LIN {X 0,Y 417.78,Z 272.398,A -85,B 0,C 180,E1 -10353.858,E2 -10353.858} C_VEL
LIN {X 0,Y 417.736,Z 275.155,A -85,B 0,C 180,E1 -10356.981,E2 -10356.981} C_VEL
LIN {X 0,Y 417.624,Z 276.659,A -85,B 0,C 180,E1 -10358.65,E2 -10358.65} C_VEL
LIN {X 0,Y 420.264,Z 284.393,A -85,B 0,C 180,E1 -10359.007,E2 -10359.007} C_VEL
LIN {X 0,Y 425.304,Z 299.305,A -85,B 0,C 180,E1 -10359.798,E2 -10359.798} C_VEL
LIN {X 0,Y 427.282,Z 306.519,A -85,B 0,C 180,E1 -10360.222,E2 -10360.222} C_VEL
LIN {X 0,Y 427.662,Z 310.082,A -85,B 0,C 180,E1 -10360.409,E2 -10360.409} C_VEL
LIN {X 0,Y 426.563,Z 315.588,A -85,B 0,C 180,E1 -10360.631,E2 -10360.631} C_VEL
LIN {X 0,Y 420.151,Z 329.943,A -85,B 0,C 180,E1 -10361.176,E2 -10361.176} C_VEL
LIN {X 0,Y 419.11,Z 333.547,A -85,B 0,C 180,E1 -10361.385,E2 -10361.385} C_VEL
LIN {X 0,Y 418.867,Z 335.334,A -85,B 0,C 180,E1 -10361.51,E2 -10361.51} C_VEL
LIN {X 0,Y 417.7,Z 349.15,A -85,B 0,C 180,E1 -10362.634,E2 -10362.634} C_VEL
LIN {X 0,Y 416.435,Z 362.009,A -85,B 0,C 180,E1 -10363.915,E2 -10363.915} C_VEL
LIN {X 0,Y 415.171,Z 374.509,A -85,B 0,C 180,E1 -10365.434,E2 -10365.434} C_VEL
LIN {X 0,Y 413.977,Z 385.392,A -85,B 0,C 180,E1 -10367.028,E2 -10367.028} C_VEL
LIN {X 0,Y 412.925,Z 394.448,A -85,B 0,C 180,E1 -10368.609,E2 -10368.609} C_VEL
LIN {X 0,Y 412.129,Z 402.506,A -85,B 0,C 180,E1 -10370.301,E2 -10370.301} C_VEL
LIN {X 0,Y 411.345,Z 410.582,A -85,B 0,C 180,E1 -10372.365,E2 -10372.365} C_VEL
LIN {X 0,Y 410.794,Z 416.403,A -85,B 0,C 180,E1 -10374.242,E2 -10374.242} C_VEL
LIN {X 0,Y 410.419,Z 421.643,A -85,B 0,C 180,E1 -10376.437,E2 -10376.437} C_VEL
LIN {X 0,Y 410.248,Z 423.698,A -85,B 0,C 180,E1 -10377.55,E2 -10377.55} C_VEL
LIN {X 0,Y 410.052,Z 425.834,A -85,B 0,C 180,E1 -10379.065,E2 -10379.065} C_VEL
LIN {X 0,Y 409.943,Z 427.623,A -85,B 0,C 180,E1 -10381.001,E2 -10381.001} C_VEL
LIN {X 0,Y 409.913,Z 428.276,A -85,B 0,C 180,E1 -10382.851,E2 -10382.851} C_VEL
LIN {X 0,Y 409.904,Z 427.963,A -85,B 0,C 180,E1 -10384.618,E2 -10384.618} C_VEL
LIN {X 0,Y 410.045,Z 426.269,A -85,B 0,C 180,E1 -10386.861,E2 -10386.861} C_VEL
LIN {X 0,Y 410.294,Z 423.778,A -85,B 0,C 180,E1 -10388.697,E2 -10388.697} C_VEL
LIN {X 0,Y 410.587,Z 420.138,A -85,B 0,C 180,E1 -10390.574,E2 -10390.574} C_VEL
LIN {X 0,Y 411.1,Z 414.621,A -85,B 0,C 180,E1 -10392.686,E2 -10392.686} C_VEL
LIN {X 0,Y 411.744,Z 407.684,A -85,B 0,C 180,E1 -10394.737,E2 -10394.737} C_VEL
LIN {X 0,Y 412.525,Z 400.757,A -85,B 0,C 180,E1 -10396.389,E2 -10396.389} C_VEL
LIN {X 0,Y 413.456,Z 392.475,A -85,B 0,C 180,E1 -10398.043,E2 -10398.043} C_VEL
LIN {X 0,Y 414.566,Z 382.455,A -85,B 0,C 180,E1 -10399.717,E2 -10399.717} C_VEL
LIN {X 0,Y 415.656,Z 372.901,A -85,B 0,C 180,E1 -10401.056,E2 -10401.056} C_VEL
LIN {X 0,Y 416.904,Z 361.556,A -85,B 0,C 180,E1 -10402.4,E2 -10402.4} C_VEL
LIN {X 0,Y 418.204,Z 348.685,A -85,B 0,C 180,E1 -10403.665,E2 -10403.665} C_VEL
LIN {X 0,Y 419.338,Z 335.97,A -85,B 0,C 180,E1 -10404.694,E2 -10404.694} C_VEL
LIN {X 0,Y 420.418,Z 322.342,A -85,B 0,C 180,E1 -10405.583,E2 -10405.583} C_VEL
LIN {X 0,Y 421.137,Z 309.245,A -85,B 0,C 180,E1 -10406.263,E2 -10406.263} C_VEL
LIN {X 0,Y 417.181,Z 296.351,A -85,B 0,C 180,E1 -10407.067,E2 -10407.067} C_VEL
LIN {X 0,Y 411.697,Z 281.87,A -85,B 0,C 180,E1 -10407.87,E2 -10407.87} C_VEL
LIN {X 0,Y 410.707,Z 278.898,A -85,B 0,C 180,E1 -10408.024,E2 -10408.024} C_VEL
LIN {X 0,Y 410.788,Z 276.178,A -85,B 0,C 180,E1 -10411.379,E2 -10411.379} C_VEL
LIN {X 0,Y 410.912,Z 273.548,A -85,B 0,C 180,E1 -10414.687,E2 -10414.687} C_VEL
LIN {X 0,Y 411.031,Z 271.058,A -85,B 0,C 180,E1 -10417.905,E2 -10417.905} C_VEL
LIN {X 0,Y 411.105,Z 269.368,A -85,B 0,C 180,E1 -10420.09,E2 -10420.09} C_VEL
LIN {X 0,Y 411.104,Z 268.906,A -85,B 0,C 180,E1 -10421.047,E2 -10421.047} C_VEL
LIN {X 0,Y 411.247,Z 268.889,A -85,B 0,C 180,E1 -10424.133,E2 -10424.133} C_VEL
LIN {X 0,Y 411.296,Z 268.878,A -85,B 0,C 180,E1 -10427.167,E2 -10427.167} C_VEL
LIN {X 0,Y 411.287,Z 268.881,A -85,B 0,C 180,E1 -10430.162,E2 -10430.162} C_VEL
LIN {X 0,Y 411.455,Z 268.86,A -85,B 0,C 180,E1 -10433.134,E2 -10433.134} C_VEL
LIN {X 0,Y 411.308,Z 268.879,A -85,B 0,C 180,E1 -10435.1,E2 -10435.1} C_VEL
LIN {X 0,Y 411.509,Z 268.851,A -85,B 0,C 180,E1 -10438.044,E2 -10438.044} C_VEL
LIN {X 0,Y 411.637,Z 268.834,A -85,B 0,C 180,E1 -10440.001,E2 -10440.001} C_VEL
LIN {X 0,Y 411.462,Z 268.859,A -85,B 0,C 180,E1 -10442.938,E2 -10442.938} C_VEL
LIN {X 0,Y 411.457,Z 268.859,A -85,B 0,C 180,E1 -10446.868,E2 -10446.868} C_VEL
LIN {X 0,Y 411.29,Z 268.88,A -85,B 0,C 180,E1 -10449.84,E2 -10449.84} C_VEL
LIN {X 0,Y 411.302,Z 268.875,A -85,B 0,C 180,E1 -10453.105,E2 -10453.105} C_VEL
LIN {X 0,Y 411.254,Z 268.882,A -85,B 0,C 180,E1 -10456.89,E2 -10456.89} C_VEL
LIN {X 0,Y 411.228,Z 268.886,A -85,B 0,C 180,E1 -10459.988,E2 -10459.988} C_VEL
LIN {X 0,Y 411.201,Z 268.89,A -85,B 0,C 180,E1 -10463.148,E2 -10463.148} C_VEL
LIN {X 0,Y 411.236,Z 268.888,A -85,B 0,C 180,E1 -10466.382,E2 -10466.382} C_VEL
LIN {X 0,Y 411.198,Z 268.895,A -85,B 0,C 180,E1 -10469.714,E2 -10469.714} C_VEL
LIN {X 0,Y 411.204,Z 268.899,A -85,B 0,C 180,E1 -10473.157,E2 -10473.157} C_VEL
LIN {X 0,Y 411.191,Z 268.898,A -85,B 0,C 180,E1 -10476.553,E2 -10476.553} C_VEL
LIN {X 0,Y 411.228,Z 269.052,A -85,B 0,C 180,E1 -10478.174,E2 -10478.174} C_VEL
LIN {X 0,Y 411.775,Z 272.063,A -85,B 0,C 180,E1 -10480.434,E2 -10480.434} C_VEL
LIN {X 0,Y 412.581,Z 276.778,A -85,B 0,C 180,E1 -10483.622,E2 -10483.622} C_VEL
LIN {X 0,Y 413.264,Z 280.257,A -85,B 0,C 180,E1 -10485.794,E2 -10485.794} C_VEL
LIN {X 0,Y 413.665,Z 283.769,A -85,B 0,C 180,E1 -10487.835,E2 -10487.835} C_VEL
LIN {X 0,Y 413.41,Z 288.694,A -85,B 0,C 180,E1 -10490.455,E2 -10490.455} C_VEL
LIN {X 0,Y 412.873,Z 294.663,A -85,B 0,C 180,E1 -10493.433,E2 -10493.433} C_VEL
LIN {X 0,Y 412.345,Z 302.105,A -85,B 0,C 180,E1 -10496.948,E2 -10496.948} C_VEL
LIN {X 0,Y 411.837,Z 310.013,A -85,B 0,C 180,E1 -10500.496,E2 -10500.496} C_VEL
LIN {X 0,Y 411.424,Z 317.27,A -85,B 0,C 180,E1 -10503.633,E2 -10503.633} C_VEL
LIN {X 0,Y 411.288,Z 320.498,A -85,B 0,C 180,E1 -10505.002,E2 -10505.002} C_VEL
LIN {X 0,Y 415.679,Z 338.456,A -85,B 0,C 180,E1 -10505.742,E2 -10505.742} C_VEL
LIN {X 0,Y 418.813,Z 353.128,A -85,B 0,C 180,E1 -10506.502,E2 -10506.502} C_VEL
LIN {X 0,Y 420.119,Z 360.598,A -85,B 0,C 180,E1 -10506.938,E2 -10506.938} C_VEL
LIN {X 0,Y 419.113,Z 374.52,A -85,B 0,C 180,E1 -10507.705,E2 -10507.705} C_VEL
LIN {X 0,Y 417.815,Z 388.486,A -85,B 0,C 180,E1 -10508.67,E2 -10508.67} C_VEL
LIN {X 0,Y 416.538,Z 401.32,A -85,B 0,C 180,E1 -10509.765,E2 -10509.765} C_VEL
LIN {X 0,Y 415.192,Z 414.332,A -85,B 0,C 180,E1 -10511.112,E2 -10511.112} C_VEL
LIN {X 0,Y 414.139,Z 425.261,A -85,B 0,C 180,E1 -10512.47,E2 -10512.47} C_VEL
LIN {X 0,Y 412.996,Z 435.377,A -85,B 0,C 180,E1 -10513.948,E2 -10513.948} C_VEL
LIN {X 0,Y 411.994,Z 445.292,A -85,B 0,C 180,E1 -10515.68,E2 -10515.68} C_VEL
LIN {X 0,Y 411.241,Z 453.581,A -85,B 0,C 180,E1 -10517.415,E2 -10517.415} C_VEL
LIN {X 0,Y 410.766,Z 460.444,A -85,B 0,C 180,E1 -10519.153,E2 -10519.153} C_VEL
LIN {X 0,Y 410.323,Z 466.793,A -85,B 0,C 180,E1 -10521.133,E2 -10521.133} C_VEL
LIN {X 0,Y 410.163,Z 471.718,A -85,B 0,C 180,E1 -10523.112,E2 -10523.112} C_VEL
LIN {X 0,Y 410.032,Z 475.329,A -85,B 0,C 180,E1 -10525.084,E2 -10525.084} C_VEL
LIN {X 0,Y 410.002,Z 477.711,A -85,B 0,C 180,E1 -10527.053,E2 -10527.053} C_VEL
LIN {X 0,Y 409.917,Z 478.915,A -85,B 0,C 180,E1 -10529.018,E2 -10529.018} C_VEL
LIN {X 0,Y 409.917,Z 478.931,A -85,B 0,C 180,E1 -10530.983,E2 -10530.983} C_VEL
LIN {X 0,Y 409.987,Z 477.754,A -85,B 0,C 180,E1 -10532.948,E2 -10532.948} C_VEL
LIN {X 0,Y 410.027,Z 475.402,A -85,B 0,C 180,E1 -10534.917,E2 -10534.917} C_VEL
LIN {X 0,Y 410.159,Z 471.832,A -85,B 0,C 180,E1 -10536.89,E2 -10536.89} C_VEL
LIN {X 0,Y 410.324,Z 466.949,A -85,B 0,C 180,E1 -10538.868,E2 -10538.868} C_VEL
LIN {X 0,Y 410.763,Z 460.638,A -85,B 0,C 180,E1 -10540.849,E2 -10540.849} C_VEL
LIN {X 0,Y 411.293,Z 453.823,A -85,B 0,C 180,E1 -10542.584,E2 -10542.584} C_VEL
LIN {X 0,Y 412,Z 445.583,A -85,B 0,C 180,E1 -10544.321,E2 -10544.321} C_VEL
LIN {X 0,Y 413.025,Z 435.723,A -85,B 0,C 180,E1 -10546.053,E2 -10546.053} C_VEL
LIN {X 0,Y 414.16,Z 425.652,A -85,B 0,C 180,E1 -10547.531,E2 -10547.531} C_VEL
LIN {X 0,Y 415.348,Z 413.696,A -85,B 0,C 180,E1 -10549.01,E2 -10549.01} C_VEL
LIN {X 0,Y 416.611,Z 401.802,A -85,B 0,C 180,E1 -10550.233,E2 -10550.233} C_VEL
LIN {X 0,Y 417.807,Z 388.969,A -85,B 0,C 180,E1 -10551.332,E2 -10551.332} C_VEL
LIN {X 0,Y 419.125,Z 375.006,A -85,B 0,C 180,E1 -10552.296,E2 -10552.296} C_VEL
LIN {X 0,Y 420.22,Z 360.344,A -85,B 0,C 180,E1 -10553.095,E2 -10553.095} C_VEL
LIN {X 0,Y 416.994,Z 344.752,A -85,B 0,C 180,E1 -10553.963,E2 -10553.963} C_VEL
LIN {X 0,Y 413.283,Z 329.145,A -85,B 0,C 180,E1 -10554.659,E2 -10554.659} C_VEL
LIN {X 0,Y 411.317,Z 321.374,A -85,B 0,C 180,E1 -10554.967,E2 -10554.967} C_VEL
LIN {X 0,Y 411.824,Z 313.102,A -85,B 0,C 180,E1 -10558.545,E2 -10558.545} C_VEL
LIN {X 0,Y 412.209,Z 306.413,A -85,B 0,C 180,E1 -10561.517,E2 -10561.517} C_VEL
LIN {X 0,Y 412.764,Z 298.457,A -85,B 0,C 180,E1 -10565.186,E2 -10565.186} C_VEL
LIN {X 0,Y 413.36,Z 291.494,A -85,B 0,C 180,E1 -10568.546,E2 -10568.546} C_VEL
LIN {X 0,Y 413.738,Z 286.906,A -85,B 0,C 180,E1 -10570.843,E2 -10570.843} C_VEL
LIN {X 0,Y 413.617,Z 282.727,A -85,B 0,C 180,E1 -10573.059,E2 -10573.059} C_VEL
LIN {X 0,Y 412.893,Z 278.02,A -85,B 0,C 180,E1 -10575.742,E2 -10575.742} C_VEL
LIN {X 0,Y 411.746,Z 271.777,A -85,B 0,C 180,E1 -10579.562,E2 -10579.562} C_VEL
LIN {X 0,Y 411.213,Z 268.89,A -85,B 0,C 180,E1 -10581.491,E2 -10581.491} C_VEL
LIN {X 0,Y 411.215,Z 268.89,A -85,B 0,C 180,E1 -10585.122,E2 -10585.122} C_VEL
LIN {X 0,Y 411.171,Z 268.895,A -85,B 0,C 180,E1 -10588.002,E2 -10588.002} C_VEL
LIN {X 0,Y 411.224,Z 268.885,A -85,B 0,C 180,E1 -10591.41,E2 -10591.41} C_VEL
LIN {X 0,Y 411.244,Z 268.882,A -85,B 0,C 180,E1 -10593.619,E2 -10593.619} C_VEL
LIN {X 0,Y 411.209,Z 268.891,A -85,B 0,C 180,E1 -10596.852,E2 -10596.852} C_VEL
LIN {X 0,Y 411.221,Z 268.885,A -85,B 0,C 180,E1 -10600.05,E2 -10600.05} C_VEL
LIN {X 0,Y 411.269,Z 268.88,A -85,B 0,C 180,E1 -10603.131,E2 -10603.131} C_VEL
LIN {X 0,Y 411.311,Z 268.877,A -85,B 0,C 180,E1 -10606.895,E2 -10606.895} C_VEL
LIN {X 0,Y 411.297,Z 268.878,A -85,B 0,C 180,E1 -10610.16,E2 -10610.16} C_VEL
LIN {X 0,Y 411.428,Z 268.859,A -85,B 0,C 180,E1 -10613.132,E2 -10613.132} C_VEL
LIN {X 0,Y 411.311,Z 268.874,A -85,B 0,C 180,E1 -10615.098,E2 -10615.098} C_VEL
LIN {X 0,Y 411.516,Z 268.85,A -85,B 0,C 180,E1 -10618.042,E2 -10618.042} C_VEL
LIN {X 0,Y 411.647,Z 268.834,A -85,B 0,C 180,E1 -10619.999,E2 -10619.999} C_VEL
LIN {X 0,Y 411.46,Z 268.856,A -85,B 0,C 180,E1 -10622.936,E2 -10622.936} C_VEL
LIN {X 0,Y 411.464,Z 268.856,A -85,B 0,C 180,E1 -10626.866,E2 -10626.866} C_VEL
LIN {X 0,Y 411.357,Z 268.869,A -85,B 0,C 180,E1 -10628.844,E2 -10628.844} C_VEL
LIN {X 0,Y 411.286,Z 268.879,A -85,B 0,C 180,E1 -10631.831,E2 -10631.831} C_VEL
LIN {X 0,Y 411.262,Z 268.88,A -85,B 0,C 180,E1 -10634.851,E2 -10634.851} C_VEL
LIN {X 0,Y 411.254,Z 268.884,A -85,B 0,C 180,E1 -10637.914,E2 -10637.914} C_VEL
LIN {X 0,Y 411.197,Z 268.888,A -85,B 0,C 180,E1 -10641.033,E2 -10641.033} C_VEL
LIN {X 0,Y 411.227,Z 268.888,A -85,B 0,C 180,E1 -10644.214,E2 -10644.214} C_VEL
LIN {X 0,Y 411.258,Z 268.881,A -85,B 0,C 180,E1 -10647.476,E2 -10647.476} C_VEL
LIN {X 0,Y 411.188,Z 268.888,A -85,B 0,C 180,E1 -10650.846,E2 -10650.846} C_VEL
LIN {X 0,Y 411.204,Z 268.89,A -85,B 0,C 180,E1 -10654.332,E2 -10654.332} C_VEL
LIN {X 0,Y 411.198,Z 268.892,A -85,B 0,C 180,E1 -10657.971,E2 -10657.971} C_VEL
LIN {X 0,Y 411.18,Z 268.891,A -85,B 0,C 180,E1 -10660.502,E2 -10660.502} C_VEL
LIN {X 0,Y 411.173,Z 268.891,A -85,B 0,C 180,E1 -10663.131,E2 -10663.131} C_VEL
LIN {X 0,Y 411.228,Z 268.889,A -85,B 0,C 180,E1 -10665.87,E2 -10665.87} C_VEL
LIN {X 0,Y 411.204,Z 268.886,A -85,B 0,C 180,E1 -10668.763,E2 -10668.763} C_VEL
LIN {X 0,Y 411.198,Z 268.891,A -85,B 0,C 180,E1 -10672.026,E2 -10672.026} C_VEL
LIN {X 0,Y 411.2,Z 268.893,A -85,B 0,C 180,E1 -10675.665,E2 -10675.665} C_VEL
LIN {X 0,Y 411.19,Z 268.89,A -85,B 0,C 180,E1 -10679.152,E2 -10679.152} C_VEL
LIN {X 0,Y 411.252,Z 268.881,A -85,B 0,C 180,E1 -10682.521,E2 -10682.521} C_VEL
LIN {X 0,Y 411.219,Z 268.889,A -85,B 0,C 180,E1 -10685.783,E2 -10685.783} C_VEL
LIN {X 0,Y 411.187,Z 268.89,A -85,B 0,C 180,E1 -10688.965,E2 -10688.965} C_VEL
LIN {X 0,Y 411.243,Z 268.883,A -85,B 0,C 180,E1 -10692.084,E2 -10692.084} C_VEL
LIN {X 0,Y 411.253,Z 268.884,A -85,B 0,C 180,E1 -10695.146,E2 -10695.146} C_VEL
LIN {X 0,Y 411.29,Z 268.876,A -85,B 0,C 180,E1 -10698.167,E2 -10698.167} C_VEL
LIN {X 0,Y 411.471,Z 268.853,A -85,B 0,C 180,E1 -10702.146,E2 -10702.146} C_VEL
LIN {X 0,Y 411.457,Z 268.855,A -85,B 0,C 180,E1 -10704.117,E2 -10704.117} C_VEL
LIN {X 0,Y 411.291,Z 269.014,A -85,B 0,C 180,E1 -10709.02,E2 -10709.02} C_VEL
LIN {X 0,Y 410.739,Z 273.276,A -85,B 0,C 180,E1 -10713.924,E2 -10713.924} C_VEL
LIN {X 0,Y 410.686,Z 275.98,A -85,B 0,C 180,E1 -10717.015,E2 -10717.015} C_VEL
LIN {X 0,Y 410.626,Z 277.162,A -85,B 0,C 180,E1 -10718.24,E2 -10718.24} C_VEL
LIN {X 0,Y 412.386,Z 282.474,A -85,B 0,C 180,E1 -10718.475,E2 -10718.475} C_VEL
LIN {X 0,Y 417.785,Z 297.852,A -85,B 0,C 180,E1 -10719.298,E2 -10719.298} C_VEL
LIN {X 0,Y 420.605,Z 307.968,A -85,B 0,C 180,E1 -10719.905,E2 -10719.905} C_VEL
LIN {X 0,Y 420.098,Z 318.721,A -85,B 0,C 180,E1 -10720.454,E2 -10720.454} C_VEL
LIN {X 0,Y 419.006,Z 333.29,A -85,B 0,C 180,E1 -10721.366,E2 -10721.366} C_VEL
LIN {X 0,Y 418.867,Z 335.334,A -85,B 0,C 180,E1 -10721.51,E2 -10721.51} C_VEL
LIN {X 0,Y 417.847,Z 340.577,A -85,B 0,C 180,E1 -10721.876,E2 -10721.876} C_VEL
LIN {X 0,Y 414.391,Z 348.97,A -85,B 0,C 180,E1 -10722.435,E2 -10722.435} C_VEL
LIN {X 0,Y 410.883,Z 357.019,A -85,B 0,C 180,E1 -10723.062,E2 -10723.062} C_VEL
LIN {X 0,Y 409.776,Z 361.712,A -85,B 0,C 180,E1 -10723.527,E2 -10723.527} C_VEL
LIN {X 0,Y 408.522,Z 373.488,A -85,B 0,C 180,E1 -10724.954,E2 -10724.954} C_VEL
LIN {X 0,Y 407.275,Z 384.421,A -85,B 0,C 180,E1 -10726.542,E2 -10726.542} C_VEL
LIN {X 0,Y 406.168,Z 393.656,A -85,B 0,C 180,E1 -10728.146,E2 -10728.146} C_VEL
LIN {X 0,Y 405.343,Z 401.462,A -85,B 0,C 180,E1 -10729.76,E2 -10729.76} C_VEL
LIN {X 0,Y 404.591,Z 408.16,A -85,B 0,C 180,E1 -10731.393,E2 -10731.393} C_VEL
LIN {X 0,Y 404.021,Z 414.137,A -85,B 0,C 180,E1 -10733.158,E2 -10733.158} C_VEL
LIN {X 0,Y 403.539,Z 419.374,A -85,B 0,C 180,E1 -10735.096,E2 -10735.096} C_VEL
LIN {X 0,Y 403.301,Z 423.199,A -85,B 0,C 180,E1 -10736.941,E2 -10736.941} C_VEL
LIN {X 0,Y 402.959,Z 426.531,A -85,B 0,C 180,E1 -10739.231,E2 -10739.231} C_VEL
LIN {X 0,Y 402.836,Z 428.356,A -85,B 0,C 180,E1 -10741.559,E2 -10741.559} C_VEL
LIN {X 0,Y 402.805,Z 428.751,A -85,B 0,C 180,E1 -10743.127,E2 -10743.127} C_VEL
LIN {X 0,Y 402.833,Z 428.189,A -85,B 0,C 180,E1 -10745.15,E2 -10745.15} C_VEL
LIN {X 0,Y 402.948,Z 427.023,A -85,B 0,C 180,E1 -10746.652,E2 -10746.652} C_VEL
LIN {X 0,Y 403.242,Z 424.131,A -85,B 0,C 180,E1 -10748.86,E2 -10748.86} C_VEL
LIN {X 0,Y 403.568,Z 420.469,A -85,B 0,C 180,E1 -10750.771,E2 -10750.771} C_VEL
LIN {X 0,Y 404.044,Z 415.487,A -85,B 0,C 180,E1 -10752.715,E2 -10752.715} C_VEL
LIN {X 0,Y 404.641,Z 409.4,A -85,B 0,C 180,E1 -10754.596,E2 -10754.596} C_VEL
LIN {X 0,Y 405.49,Z 402.426,A -85,B 0,C 180,E1 -10756.349,E2 -10756.349} C_VEL
LIN {X 0,Y 406.423,Z 394.39,A -85,B 0,C 180,E1 -10758.035,E2 -10758.035} C_VEL
LIN {X 0,Y 407.543,Z 384.675,A -85,B 0,C 180,E1 -10759.735,E2 -10759.735} C_VEL
LIN {X 0,Y 408.826,Z 374.222,A -85,B 0,C 180,E1 -10761.26,E2 -10761.26} C_VEL
LIN {X 0,Y 410.137,Z 363.075,A -85,B 0,C 180,E1 -10762.623,E2 -10762.623} C_VEL
LIN {X 0,Y 411.448,Z 350.593,A -85,B 0,C 180,E1 -10763.895,E2 -10763.895} C_VEL
LIN {X 0,Y 412.66,Z 337.723,A -85,B 0,C 180,E1 -10764.973,E2 -10764.973} C_VEL
LIN {X 0,Y 413.849,Z 323.666,A -85,B 0,C 180,E1 -10765.918,E2 -10765.918} C_VEL
LIN {X 0,Y 414.655,Z 311.283,A -85,B 0,C 180,E1 -10766.576,E2 -10766.576} C_VEL
LIN {X 0,Y 410.865,Z 298.721,A -85,B 0,C 180,E1 -10767.398,E2 -10767.398} C_VEL
LIN {X 0,Y 405.94,Z 285.386,A -85,B 0,C 180,E1 -10768.187,E2 -10768.187} C_VEL
LIN {X 0,Y 403.832,Z 280.278,A -85,B 0,C 180,E1 -10768.463,E2 -10768.463} C_VEL
LIN {X 0,Y 403.678,Z 279.406,A -85,B 0,C 180,E1 -10768.515,E2 -10768.515} C_VEL
LIN {X 0,Y 403.788,Z 276.656,A -85,B 0,C 180,E1 -10771.971,E2 -10771.971} C_VEL
LIN {X 0,Y 403.902,Z 274.043,A -85,B 0,C 180,E1 -10775.318,E2 -10775.318} C_VEL
LIN {X 0,Y 404.017,Z 271.536,A -85,B 0,C 180,E1 -10778.575,E2 -10778.575} C_VEL
LIN {X 0,Y 404.056,Z 269.973,A -85,B 0,C 180,E1 -10780.704,E2 -10780.704} C_VEL
LIN {X 0,Y 404.213,Z 269.765,A -85,B 0,C 180,E1 -10783.849,E2 -10783.849} C_VEL
LIN {X 0,Y 404.275,Z 269.753,A -85,B 0,C 180,E1 -10786.94,E2 -10786.94} C_VEL
LIN {X 0,Y 404.252,Z 269.757,A -85,B 0,C 180,E1 -10789.989,E2 -10789.989} C_VEL
LIN {X 0,Y 404.406,Z 269.737,A -85,B 0,C 180,E1 -10793.014,E2 -10793.014} C_VEL
LIN {X 0,Y 404.28,Z 269.754,A -85,B 0,C 180,E1 -10795.015,E2 -10795.015} C_VEL
LIN {X 0,Y 404.478,Z 269.726,A -85,B 0,C 180,E1 -10798.01,E2 -10798.01} C_VEL
LIN {X 0,Y 404.607,Z 269.71,A -85,B 0,C 180,E1 -10800.001,E2 -10800.001} C_VEL
LIN {X 0,Y 404.419,Z 269.736,A -85,B 0,C 180,E1 -10802.989,E2 -10802.989} C_VEL
LIN {X 0,Y 404.408,Z 269.738,A -85,B 0,C 180,E1 -10806.988,E2 -10806.988} C_VEL
LIN {X 0,Y 404.255,Z 269.755,A -85,B 0,C 180,E1 -10810.013,E2 -10810.013} C_VEL
LIN {X 0,Y 404.263,Z 269.752,A -85,B 0,C 180,E1 -10813.212,E2 -10813.212} C_VEL
LIN {X 0,Y 404.212,Z 269.758,A -85,B 0,C 180,E1 -10817.008,E2 -10817.008} C_VEL
LIN {X 0,Y 404.161,Z 269.768,A -85,B 0,C 180,E1 -10820.353,E2 -10820.353} C_VEL
LIN {X 0,Y 404.167,Z 269.765,A -85,B 0,C 180,E1 -10823.575,E2 -10823.575} C_VEL
LIN {X 0,Y 404.181,Z 269.764,A -85,B 0,C 180,E1 -10825.767,E2 -10825.767} C_VEL
LIN {X 0,Y 404.193,Z 269.766,A -85,B 0,C 180,E1 -10828.001,E2 -10828.001} C_VEL
LIN {X 0,Y 404.137,Z 269.777,A -85,B 0,C 180,E1 -10831.559,E2 -10831.559} C_VEL
LIN {X 0,Y 404.182,Z 269.772,A -85,B 0,C 180,E1 -10835.017,E2 -10835.017} C_VEL
LIN {X 0,Y 404.14,Z 269.806,A -85,B 0,C 180,E1 -10837.493,E2 -10837.493} C_VEL
LIN {X 0,Y 404.816,Z 273.26,A -85,B 0,C 180,E1 -10840.194,E2 -10840.194} C_VEL
LIN {X 0,Y 405.701,Z 278.607,A -85,B 0,C 180,E1 -10843.863,E2 -10843.863} C_VEL
LIN {X 0,Y 406.495,Z 282.927,A -85,B 0,C 180,E1 -10846.565,E2 -10846.565} C_VEL
LIN {X 0,Y 406.696,Z 285.38,A -85,B 0,C 180,E1 -10847.994,E2 -10847.994} C_VEL
LIN {X 0,Y 406.443,Z 289.501,A -85,B 0,C 180,E1 -10850.225,E2 -10850.225} C_VEL
LIN {X 0,Y 405.876,Z 295.661,A -85,B 0,C 180,E1 -10853.355,E2 -10853.355} C_VEL
LIN {X 0,Y 405.325,Z 303,A -85,B 0,C 180,E1 -10856.903,E2 -10856.903} C_VEL
LIN {X 0,Y 404.813,Z 310.259,A -85,B 0,C 180,E1 -10860.234,E2 -10860.234} C_VEL
LIN {X 0,Y 404.356,Z 318.077,A -85,B 0,C 180,E1 -10863.692,E2 -10863.692} C_VEL
LIN {X 0,Y 404.275,Z 319.984,A -85,B 0,C 180,E1 -10864.518,E2 -10864.518} C_VEL
LIN {X 0,Y 408.798,Z 338.247,A -85,B 0,C 180,E1 -10865.305,E2 -10865.305} C_VEL
LIN {X 0,Y 412.078,Z 354.003,A -85,B 0,C 180,E1 -10866.146,E2 -10866.146} C_VEL
LIN {X 0,Y 413.482,Z 361.568,A -85,B 0,C 180,E1 -10866.614,E2 -10866.614} C_VEL
LIN {X 0,Y 412.359,Z 376.097,A -85,B 0,C 180,E1 -10867.452,E2 -10867.452} C_VEL
LIN {X 0,Y 410.996,Z 389.63,A -85,B 0,C 180,E1 -10868.43,E2 -10868.43} C_VEL
LIN {X 0,Y 409.549,Z 403.471,A -85,B 0,C 180,E1 -10869.667,E2 -10869.667} C_VEL
LIN {X 0,Y 408.17,Z 416.435,A -85,B 0,C 180,E1 -10871.084,E2 -10871.084} C_VEL
LIN {X 0,Y 406.849,Z 428.393,A -85,B 0,C 180,E1 -10872.664,E2 -10872.664} C_VEL
LIN {X 0,Y 405.608,Z 439.395,A -85,B 0,C 180,E1 -10874.422,E2 -10874.422} C_VEL
LIN {X 0,Y 404.685,Z 448.581,A -85,B 0,C 180,E1 -10876.186,E2 -10876.186} C_VEL
LIN {X 0,Y 404.001,Z 456.21,A -85,B 0,C 180,E1 -10877.952,E2 -10877.952} C_VEL
LIN {X 0,Y 403.573,Z 461.693,A -85,B 0,C 180,E1 -10879.465,E2 -10879.465} C_VEL
LIN {X 0,Y 403.177,Z 467.69,A -85,B 0,C 180,E1 -10881.48,E2 -10881.48} C_VEL
LIN {X 0,Y 403.058,Z 472.632,A -85,B 0,C 180,E1 -10883.667,E2 -10883.667} C_VEL
LIN {X 0,Y 402.945,Z 474.883,A -85,B 0,C 180,E1 -10884.998,E2 -10884.998} C_VEL
LIN {X 0,Y 402.903,Z 477.27,A -85,B 0,C 180,E1 -10887.001,E2 -10887.001} C_VEL
LIN {X 0,Y 402.846,Z 478.478,A -85,B 0,C 180,E1 -10889.001,E2 -10889.001} C_VEL
LIN {X 0,Y 402.846,Z 478.497,A -85,B 0,C 180,E1 -10891,E2 -10891} C_VEL
LIN {X 0,Y 402.888,Z 477.321,A -85,B 0,C 180,E1 -10893,E2 -10893} C_VEL
LIN {X 0,Y 402.938,Z 474.97,A -85,B 0,C 180,E1 -10895.004,E2 -10895.004} C_VEL
LIN {X 0,Y 403.069,Z 471.4,A -85,B 0,C 180,E1 -10897.011,E2 -10897.011} C_VEL
LIN {X 0,Y 403.266,Z 466.518,A -85,B 0,C 180,E1 -10899.025,E2 -10899.025} C_VEL
LIN {X 0,Y 403.75,Z 460.206,A -85,B 0,C 180,E1 -10901.04,E2 -10901.04} C_VEL
LIN {X 0,Y 404.306,Z 452.275,A -85,B 0,C 180,E1 -10903.061,E2 -10903.061} C_VEL
LIN {X 0,Y 405.202,Z 443.861,A -85,B 0,C 180,E1 -10904.823,E2 -10904.823} C_VEL
LIN {X 0,Y 406.266,Z 433.731,A -85,B 0,C 180,E1 -10906.585,E2 -10906.585} C_VEL
LIN {X 0,Y 407.484,Z 423.402,A -85,B 0,C 180,E1 -10908.087,E2 -10908.087} C_VEL
LIN {X 0,Y 408.812,Z 411.085,A -85,B 0,C 180,E1 -10909.587,E2 -10909.587} C_VEL
LIN {X 0,Y 410.289,Z 397.384,A -85,B 0,C 180,E1 -10910.952,E2 -10910.952} C_VEL
LIN {X 0,Y 411.479,Z 385.335,A -85,B 0,C 180,E1 -10911.94,E2 -10911.94} C_VEL
LIN {X 0,Y 412.867,Z 370.563,A -85,B 0,C 180,E1 -10912.917,E2 -10912.917} C_VEL
LIN {X 0,Y 413.542,Z 361.493,A -85,B 0,C 180,E1 -10913.406,E2 -10913.406} C_VEL
LIN {X 0,Y 410.433,Z 346.117,A -85,B 0,C 180,E1 -10914.299,E2 -10914.299} C_VEL
LIN {X 0,Y 406.761,Z 330.482,A -85,B 0,C 180,E1 -10915.034,E2 -10915.034} C_VEL
LIN {X 0,Y 404.327,Z 320.975,A -85,B 0,C 180,E1 -10915.423,E2 -10915.423} C_VEL
LIN {X 0,Y 404.752,Z 313.952,A -85,B 0,C 180,E1 -10918.523,E2 -10918.523} C_VEL
LIN {X 0,Y 405.136,Z 307.697,A -85,B 0,C 180,E1 -10921.361,E2 -10921.361} C_VEL
LIN {X 0,Y 405.698,Z 300.193,A -85,B 0,C 180,E1 -10924.867,E2 -10924.867} C_VEL
LIN {X 0,Y 406.219,Z 293.982,A -85,B 0,C 180,E1 -10927.893,E2 -10927.893} C_VEL
LIN {X 0,Y 406.681,Z 288.843,A -85,B 0,C 180,E1 -10930.502,E2 -10930.502} C_VEL
LIN {X 0,Y 406.744,Z 285.309,A -85,B 0,C 180,E1 -10932.367,E2 -10932.367} C_VEL
LIN {X 0,Y 406.2,Z 280.997,A -85,B 0,C 180,E1 -10934.815,E2 -10934.815} C_VEL
LIN {X 0,Y 405.171,Z 275.348,A -85,B 0,C 180,E1 -10938.235,E2 -10938.235} C_VEL
LIN {X 0,Y 404.228,Z 270.018,A -85,B 0,C 180,E1 -10941.725,E2 -10941.725} C_VEL
LIN {X 0,Y 404.147,Z 269.77,A -85,B 0,C 180,E1 -10942.508,E2 -10942.508} C_VEL
LIN {X 0,Y 404.189,Z 269.765,A -85,B 0,C 180,E1 -10944.984,E2 -10944.984} C_VEL
LIN {X 0,Y 404.147,Z 269.769,A -85,B 0,C 180,E1 -10948.553,E2 -10948.553} C_VEL
LIN {X 0,Y 404.201,Z 269.759,A -85,B 0,C 180,E1 -10952,E2 -10952} C_VEL
LIN {X 0,Y 404.183,Z 269.762,A -85,B 0,C 180,E1 -10955.334,E2 -10955.334} C_VEL
LIN {X 0,Y 404.145,Z 269.771,A -85,B 0,C 180,E1 -10958.58,E2 -10958.58} C_VEL
LIN {X 0,Y 404.216,Z 269.757,A -85,B 0,C 180,E1 -10961.761,E2 -10961.761} C_VEL
LIN {X 0,Y 404.212,Z 269.761,A -85,B 0,C 180,E1 -10964.881,E2 -10964.881} C_VEL
LIN {X 0,Y 404.261,Z 269.752,A -85,B 0,C 180,E1 -10967.958,E2 -10967.958} C_VEL
LIN {X 0,Y 404.294,Z 269.749,A -85,B 0,C 180,E1 -10970.998,E2 -10970.998} C_VEL
LIN {X 0,Y 404.397,Z 269.736,A -85,B 0,C 180,E1 -10974.014,E2 -10974.014} C_VEL
LIN {X 0,Y 404.485,Z 269.725,A -85,B 0,C 180,E1 -10978.008,E2 -10978.008} C_VEL
LIN {X 0,Y 404.616,Z 269.709,A -85,B 0,C 180,E1 -10979.999,E2 -10979.999} C_VEL
LIN {X 0,Y 404.418,Z 269.733,A -85,B 0,C 180,E1 -10982.987,E2 -10982.987} C_VEL
LIN {X 0,Y 404.415,Z 269.733,A -85,B 0,C 180,E1 -10986.986,E2 -10986.986} C_VEL
LIN {X 0,Y 404.261,Z 269.755,A -85,B 0,C 180,E1 -10990.01,E2 -10990.01} C_VEL
LIN {X 0,Y 404.269,Z 269.75,A -85,B 0,C 180,E1 -10993.21,E2 -10993.21} C_VEL
LIN {X 0,Y 404.217,Z 269.757,A -85,B 0,C 180,E1 -10997.006,E2 -10997.006} C_VEL
LIN {X 0,Y 404.165,Z 269.768,A -85,B 0,C 180,E1 -11000.35,E2 -11000.35} C_VEL
LIN {X 0,Y 404.17,Z 269.764,A -85,B 0,C 180,E1 -11003.573,E2 -11003.573} C_VEL
LIN {X 0,Y 404.183,Z 269.764,A -85,B 0,C 180,E1 -11005.765,E2 -11005.765} C_VEL
LIN {X 0,Y 404.194,Z 269.765,A -85,B 0,C 180,E1 -11007.998,E2 -11007.998} C_VEL
LIN {X 0,Y 404.137,Z 269.768,A -85,B 0,C 180,E1 -11011.556,E2 -11011.556} C_VEL
LIN {X 0,Y 404.183,Z 269.761,A -85,B 0,C 180,E1 -11015.014,E2 -11015.014} C_VEL
LIN {X 0,Y 404.156,Z 269.765,A -85,B 0,C 180,E1 -11018.755,E2 -11018.755} C_VEL
LIN {X 0,Y 404.121,Z 269.773,A -85,B 0,C 180,E1 -11021.598,E2 -11021.598} C_VEL
LIN {X 0,Y 404.152,Z 269.765,A -85,B 0,C 180,E1 -11024.522,E2 -11024.522} C_VEL
LIN {X 0,Y 404.203,Z 269.76,A -85,B 0,C 180,E1 -11027.304,E2 -11027.304} C_VEL
LIN {X 0,Y 404.163,Z 269.768,A -85,B 0,C 180,E1 -11029.954,E2 -11029.954} C_VEL
LIN {X 0,Y 404.134,Z 269.768,A -85,B 0,C 180,E1 -11033.123,E2 -11033.123} C_VEL
LIN {X 0,Y 404.138,Z 269.768,A -85,B 0,C 180,E1 -11036.186,E2 -11036.186} C_VEL
LIN {X 0,Y 404.146,Z 269.771,A -85,B 0,C 180,E1 -11039.714,E2 -11039.714} C_VEL
LIN {X 0,Y 404.187,Z 269.762,A -85,B 0,C 180,E1 -11043.122,E2 -11043.122} C_VEL
LIN {X 0,Y 404.169,Z 269.767,A -85,B 0,C 180,E1 -11045.333,E2 -11045.333} C_VEL
LIN {X 0,Y 404.13,Z 269.767,A -85,B 0,C 180,E1 -11048.579,E2 -11048.579} C_VEL
LIN {X 0,Y 404.201,Z 269.763,A -85,B 0,C 180,E1 -11051.761,E2 -11051.761} C_VEL
LIN {X 0,Y 404.198,Z 269.761,A -85,B 0,C 180,E1 -11054.881,E2 -11054.881} C_VEL
LIN {X 0,Y 404.26,Z 269.753,A -85,B 0,C 180,E1 -11057.958,E2 -11057.958} C_VEL
LIN {X 0,Y 404.422,Z 269.731,A -85,B 0,C 180,E1 -11062.099,E2 -11062.099} C_VEL
LIN {X 0,Y 404.406,Z 269.733,A -85,B 0,C 180,E1 -11064.014,E2 -11064.014} C_VEL
LIN {X 0,Y 404.259,Z 269.868,A -85,B 0,C 180,E1 -11069.003,E2 -11069.003} C_VEL
LIN {X 0,Y 403.698,Z 274.152,A -85,B 0,C 180,E1 -11073.992,E2 -11073.992} C_VEL
LIN {X 0,Y 403.579,Z 277.489,A -85,B 0,C 180,E1 -11077.785,E2 -11077.785} C_VEL
LIN {X 0,Y 406.476,Z 285.803,A -85,B 0,C 180,E1 -11078.184,E2 -11078.184} C_VEL
LIN {X 0,Y 411.618,Z 300.889,A -85,B 0,C 180,E1 -11079.04,E2 -11079.04} C_VEL
LIN {X 0,Y 414.121,Z 310.133,A -85,B 0,C 180,E1 -11079.627,E2 -11079.627} C_VEL
LIN {X 0,Y 413.15,Z 324.594,A -85,B 0,C 180,E1 -11080.412,E2 -11080.412} C_VEL
LIN {X 0,Y 412.088,Z 337.678,A -85,B 0,C 180,E1 -11081.31,E2 -11081.31} C_VEL
LIN {X 0,Y 410.944,Z 350.487,A -85,B 0,C 180,E1 -11082.391,E2 -11082.391} C_VEL
LIN {X 0,Y 409.776,Z 361.712,A -85,B 0,C 180,E1 -11083.527,E2 -11083.527} C_VEL
LIN {X 0,Y 408.672,Z 366.345,A -85,B 0,C 180,E1 -11084.021,E2 -11084.021} C_VEL
LIN {X 0,Y 405.115,Z 373.747,A -85,B 0,C 180,E1 -11084.811,E2 -11084.811} C_VEL
LIN {X 0,Y 401.552,Z 380.799,A -85,B 0,C 180,E1 -11085.667,E2 -11085.667} C_VEL
LIN {X 0,Y 400.443,Z 384.781,A -85,B 0,C 180,E1 -11086.258,E2 -11086.258} C_VEL
LIN {X 0,Y 399.181,Z 394.969,A -85,B 0,C 180,E1 -11088.067,E2 -11088.067} C_VEL
LIN {X 0,Y 398.262,Z 403.178,A -85,B 0,C 180,E1 -11089.836,E2 -11089.836} C_VEL
LIN {X 0,Y 397.426,Z 410.692,A -85,B 0,C 180,E1 -11091.799,E2 -11091.799} C_VEL
LIN {X 0,Y 396.833,Z 415.962,A -85,B 0,C 180,E1 -11093.482,E2 -11093.482} C_VEL
LIN {X 0,Y 396.438,Z 420.589,A -85,B 0,C 180,E1 -11095.299,E2 -11095.299} C_VEL
LIN {X 0,Y 396.12,Z 424.754,A -85,B 0,C 180,E1 -11097.492,E2 -11097.492} C_VEL
LIN {X 0,Y 395.819,Z 427.636,A -85,B 0,C 180,E1 -11099.811,E2 -11099.811} C_VEL
LIN {X 0,Y 395.77,Z 428.789,A -85,B 0,C 180,E1 -11101.532,E2 -11101.532} C_VEL
LIN {X 0,Y 395.732,Z 429.158,A -85,B 0,C 180,E1 -11103.419,E2 -11103.419} C_VEL
LIN {X 0,Y 395.77,Z 428.62,A -85,B 0,C 180,E1 -11105.231,E2 -11105.231} C_VEL
LIN {X 0,Y 395.919,Z 427.05,A -85,B 0,C 180,E1 -11107.123,E2 -11107.123} C_VEL
LIN {X 0,Y 396.146,Z 425.054,A -85,B 0,C 180,E1 -11108.687,E2 -11108.687} C_VEL
LIN {X 0,Y 396.542,Z 420.791,A -85,B 0,C 180,E1 -11110.976,E2 -11110.976} C_VEL
LIN {X 0,Y 397.041,Z 415.954,A -85,B 0,C 180,E1 -11112.892,E2 -11112.892} C_VEL
LIN {X 0,Y 397.796,Z 409.069,A -85,B 0,C 180,E1 -11115.036,E2 -11115.036} C_VEL
LIN {X 0,Y 398.83,Z 400.824,A -85,B 0,C 180,E1 -11117.073,E2 -11117.073} C_VEL
LIN {X 0,Y 399.883,Z 392.41,A -85,B 0,C 180,E1 -11118.776,E2 -11118.776} C_VEL
LIN {X 0,Y 401.089,Z 382.596,A -85,B 0,C 180,E1 -11120.441,E2 -11120.441} C_VEL
LIN {X 0,Y 402.434,Z 371.844,A -85,B 0,C 180,E1 -11121.961,E2 -11121.961} C_VEL
LIN {X 0,Y 403.863,Z 360.4,A -85,B 0,C 180,E1 -11123.311,E2 -11123.311} C_VEL
LIN {X 0,Y 405.222,Z 347.281,A -85,B 0,C 180,E1 -11124.6,E2 -11124.6} C_VEL
LIN {X 0,Y 406.505,Z 334.294,A -85,B 0,C 180,E1 -11125.636,E2 -11125.636} C_VEL
LIN {X 0,Y 407.713,Z 319.434,A -85,B 0,C 180,E1 -11126.582,E2 -11126.582} C_VEL
LIN {X 0,Y 408.059,Z 312.328,A -85,B 0,C 180,E1 -11126.962,E2 -11126.962} C_VEL
LIN {X 0,Y 403.59,Z 298.047,A -85,B 0,C 180,E1 -11127.933,E2 -11127.933} C_VEL
LIN {X 0,Y 398.715,Z 285.478,A -85,B 0,C 180,E1 -11128.706,E2 -11128.706} C_VEL
LIN {X 0,Y 396.682,Z 280.322,A -85,B 0,C 180,E1 -11128.988,E2 -11128.988} C_VEL
LIN {X 0,Y 396.641,Z 279.908,A -85,B 0,C 180,E1 -11129.033,E2 -11129.033} C_VEL
LIN {X 0,Y 396.802,Z 277.114,A -85,B 0,C 180,E1 -11132.582,E2 -11132.582} C_VEL
LIN {X 0,Y 396.885,Z 274.53,A -85,B 0,C 180,E1 -11135.967,E2 -11135.967} C_VEL
LIN {X 0,Y 397.007,Z 272.081,A -85,B 0,C 180,E1 -11139.266,E2 -11139.266} C_VEL
LIN {X 0,Y 397.018,Z 270.662,A -85,B 0,C 180,E1 -11141.421,E2 -11141.421} C_VEL
LIN {X 0,Y 397.158,Z 270.644,A -85,B 0,C 180,E1 -11143.554,E2 -11143.554} C_VEL
LIN {X 0,Y 397.221,Z 270.633,A -85,B 0,C 180,E1 -11146.704,E2 -11146.704} C_VEL
LIN {X 0,Y 397.212,Z 270.634,A -85,B 0,C 180,E1 -11149.81,E2 -11149.81} C_VEL
LIN {X 0,Y 397.358,Z 270.615,A -85,B 0,C 180,E1 -11152.889,E2 -11152.889} C_VEL
LIN {X 0,Y 397.251,Z 270.629,A -85,B 0,C 180,E1 -11154.926,E2 -11154.926} C_VEL
LIN {X 0,Y 397.447,Z 270.602,A -85,B 0,C 180,E1 -11157.974,E2 -11157.974} C_VEL
LIN {X 0,Y 397.576,Z 270.585,A -85,B 0,C 180,E1 -11160.001,E2 -11160.001} C_VEL
LIN {X 0,Y 397.377,Z 270.613,A -85,B 0,C 180,E1 -11163.042,E2 -11163.042} C_VEL
LIN {X 0,Y 397.36,Z 270.615,A -85,B 0,C 180,E1 -11167.113,E2 -11167.113} C_VEL
LIN {X 0,Y 397.215,Z 270.631,A -85,B 0,C 180,E1 -11170.192,E2 -11170.192} C_VEL
LIN {X 0,Y 397.223,Z 270.629,A -85,B 0,C 180,E1 -11173.322,E2 -11173.322} C_VEL
LIN {X 0,Y 397.179,Z 270.634,A -85,B 0,C 180,E1 -11177.156,E2 -11177.156} C_VEL
LIN {X 0,Y 397.1,Z 270.647,A -85,B 0,C 180,E1 -11180.731,E2 -11180.731} C_VEL
LIN {X 0,Y 397.131,Z 270.643,A -85,B 0,C 180,E1 -11184.019,E2 -11184.019} C_VEL
LIN {X 0,Y 397.192,Z 270.634,A -85,B 0,C 180,E1 -11187.391,E2 -11187.391} C_VEL
LIN {X 0,Y 397.076,Z 270.653,A -85,B 0,C 180,E1 -11190.883,E2 -11190.883} C_VEL
LIN {X 0,Y 397.123,Z 270.653,A -85,B 0,C 180,E1 -11194.494,E2 -11194.494} C_VEL
LIN {X 0,Y 397.112,Z 270.806,A -85,B 0,C 180,E1 -11196.994,E2 -11196.994} C_VEL
LIN {X 0,Y 397.716,Z 273.913,A -85,B 0,C 180,E1 -11199.506,E2 -11199.506} C_VEL
LIN {X 0,Y 398.293,Z 277.575,A -85,B 0,C 180,E1 -11202.176,E2 -11202.176} C_VEL
LIN {X 0,Y 399.199,Z 282.147,A -85,B 0,C 180,E1 -11205.235,E2 -11205.235} C_VEL
LIN {X 0,Y 399.705,Z 286.025,A -85,B 0,C 180,E1 -11207.603,E2 -11207.603} C_VEL
LIN {X 0,Y 399.476,Z 290.417,A -85,B 0,C 180,E1 -11210.049,E2 -11210.049} C_VEL
LIN {X 0,Y 398.885,Z 296.475,A -85,B 0,C 180,E1 -11213.199,E2 -11213.199} C_VEL
LIN {X 0,Y 398.295,Z 303.848,A -85,B 0,C 180,E1 -11216.839,E2 -11216.839} C_VEL
LIN {X 0,Y 397.734,Z 311.323,A -85,B 0,C 180,E1 -11220.347,E2 -11220.347} C_VEL
LIN {X 0,Y 397.291,Z 318.887,A -85,B 0,C 180,E1 -11223.754,E2 -11223.754} C_VEL
LIN {X 0,Y 397.253,Z 319.628,A -85,B 0,C 180,E1 -11224.033,E2 -11224.033} C_VEL
LIN {X 0,Y 401.597,Z 336.308,A -85,B 0,C 180,E1 -11224.776,E2 -11224.776} C_VEL
LIN {X 0,Y 404.803,Z 352.171,A -85,B 0,C 180,E1 -11225.62,E2 -11225.62} C_VEL
LIN {X 0,Y 406.83,Z 362.642,A -85,B 0,C 180,E1 -11226.289,E2 -11226.289} C_VEL
LIN {X 0,Y 405.731,Z 376.185,A -85,B 0,C 180,E1 -11227.093,E2 -11227.093} C_VEL
LIN {X 0,Y 404.214,Z 390.778,A -85,B 0,C 180,E1 -11228.184,E2 -11228.184} C_VEL
LIN {X 0,Y 402.697,Z 404.288,A -85,B 0,C 180,E1 -11229.438,E2 -11229.438} C_VEL
LIN {X 0,Y 401.331,Z 416.243,A -85,B 0,C 180,E1 -11230.781,E2 -11230.781} C_VEL
LIN {X 0,Y 400.015,Z 427.937,A -85,B 0,C 180,E1 -11232.359,E2 -11232.359} C_VEL
LIN {X 0,Y 398.677,Z 438.937,A -85,B 0,C 180,E1 -11234.144,E2 -11234.144} C_VEL
LIN {X 0,Y 397.679,Z 448.235,A -85,B 0,C 180,E1 -11235.963,E2 -11235.963} C_VEL
LIN {X 0,Y 396.977,Z 455.748,A -85,B 0,C 180,E1 -11237.735,E2 -11237.735} C_VEL
LIN {X 0,Y 396.529,Z 461.234,A -85,B 0,C 180,E1 -11239.275,E2 -11239.275} C_VEL
LIN {X 0,Y 396.118,Z 467.236,A -85,B 0,C 180,E1 -11241.327,E2 -11241.327} C_VEL
LIN {X 0,Y 395.989,Z 470.815,A -85,B 0,C 180,E1 -11242.864,E2 -11242.864} C_VEL
LIN {X 0,Y 395.862,Z 474.437,A -85,B 0,C 180,E1 -11244.908,E2 -11244.908} C_VEL
LIN {X 0,Y 395.805,Z 476.828,A -85,B 0,C 180,E1 -11246.947,E2 -11246.947} C_VEL
LIN {X 0,Y 395.776,Z 478.041,A -85,B 0,C 180,E1 -11248.983,E2 -11248.983} C_VEL
LIN {X 0,Y 395.777,Z 478.063,A -85,B 0,C 180,E1 -11251.018,E2 -11251.018} C_VEL
LIN {X 0,Y 395.791,Z 476.886,A -85,B 0,C 180,E1 -11253.054,E2 -11253.054} C_VEL
LIN {X 0,Y 395.855,Z 474.537,A -85,B 0,C 180,E1 -11255.094,E2 -11255.094} C_VEL
LIN {X 0,Y 395.988,Z 470.965,A -85,B 0,C 180,E1 -11257.137,E2 -11257.137} C_VEL
LIN {X 0,Y 396.198,Z 466.08,A -85,B 0,C 180,E1 -11259.187,E2 -11259.187} C_VEL
LIN {X 0,Y 396.707,Z 459.765,A -85,B 0,C 180,E1 -11261.238,E2 -11261.238} C_VEL
LIN {X 0,Y 397.319,Z 451.833,A -85,B 0,C 180,E1 -11263.295,E2 -11263.295} C_VEL
LIN {X 0,Y 398.248,Z 443.416,A -85,B 0,C 180,E1 -11265.088,E2 -11265.088} C_VEL
LIN {X 0,Y 399.37,Z 433.277,A -85,B 0,C 180,E1 -11266.88,E2 -11266.88} C_VEL
LIN {X 0,Y 400.655,Z 422.942,A -85,B 0,C 180,E1 -11268.406,E2 -11268.406} C_VEL
LIN {X 0,Y 402.012,Z 410.607,A -85,B 0,C 180,E1 -11269.932,E2 -11269.932} C_VEL
LIN {X 0,Y 403.449,Z 398.266,A -85,B 0,C 180,E1 -11271.191,E2 -11271.191} C_VEL
LIN {X 0,Y 404.876,Z 384.841,A -85,B 0,C 180,E1 -11272.317,E2 -11272.317} C_VEL
LIN {X 0,Y 406.301,Z 369.955,A -85,B 0,C 180,E1 -11273.316,E2 -11273.316} C_VEL
LIN {X 0,Y 406.876,Z 362.568,A -85,B 0,C 180,E1 -11273.726,E2 -11273.726} C_VEL
LIN {X 0,Y 403.706,Z 346.696,A -85,B 0,C 180,E1 -11274.684,E2 -11274.684} C_VEL
LIN {X 0,Y 399.945,Z 330.716,A -85,B 0,C 180,E1 -11275.464,E2 -11275.464} C_VEL
LIN {X 0,Y 397.329,Z 320.587,A -85,B 0,C 180,E1 -11275.882,E2 -11275.882} C_VEL
LIN {X 0,Y 397.868,Z 312.3,A -85,B 0,C 180,E1 -11279.644,E2 -11279.644} C_VEL
LIN {X 0,Y 398.361,Z 304.805,A -85,B 0,C 180,E1 -11283.156,E2 -11283.156} C_VEL
LIN {X 0,Y 399.025,Z 297.326,A -85,B 0,C 180,E1 -11286.787,E2 -11286.787} C_VEL
LIN {X 0,Y 399.609,Z 291.161,A -85,B 0,C 180,E1 -11289.937,E2 -11289.937} C_VEL
LIN {X 0,Y 399.766,Z 286.56,A -85,B 0,C 180,E1 -11292.406,E2 -11292.406} C_VEL
LIN {X 0,Y 399.27,Z 282.462,A -85,B 0,C 180,E1 -11294.756,E2 -11294.756} C_VEL
LIN {X 0,Y 398.164,Z 276.319,A -85,B 0,C 180,E1 -11298.553,E2 -11298.553} C_VEL
LIN {X 0,Y 397.115,Z 270.722,A -85,B 0,C 180,E1 -11302.305,E2 -11302.305} C_VEL
LIN {X 0,Y 397.13,Z 270.644,A -85,B 0,C 180,E1 -11305.506,E2 -11305.506} C_VEL
LIN {X 0,Y 397.084,Z 270.649,A -85,B 0,C 180,E1 -11309.117,E2 -11309.117} C_VEL
LIN {X 0,Y 397.2,Z 270.635,A -85,B 0,C 180,E1 -11312.609,E2 -11312.609} C_VEL
LIN {X 0,Y 397.139,Z 270.638,A -85,B 0,C 180,E1 -11315.981,E2 -11315.981} C_VEL
LIN {X 0,Y 397.145,Z 270.637,A -85,B 0,C 180,E1 -11319.704,E2 -11319.704} C_VEL
LIN {X 0,Y 397.188,Z 270.637,A -85,B 0,C 180,E1 -11322.844,E2 -11322.844} C_VEL
LIN {X 0,Y 397.234,Z 270.631,A -85,B 0,C 180,E1 -11326.702,E2 -11326.702} C_VEL
LIN {X 0,Y 397.222,Z 270.628,A -85,B 0,C 180,E1 -11329.808,E2 -11329.808} C_VEL
LIN {X 0,Y 397.323,Z 270.618,A -85,B 0,C 180,E1 -11332.886,E2 -11332.886} C_VEL
LIN {X 0,Y 397.252,Z 270.626,A -85,B 0,C 180,E1 -11334.924,E2 -11334.924} C_VEL
LIN {X 0,Y 397.454,Z 270.601,A -85,B 0,C 180,E1 -11337.972,E2 -11337.972} C_VEL
LIN {X 0,Y 397.585,Z 270.585,A -85,B 0,C 180,E1 -11339.999,E2 -11339.999} C_VEL
LIN {X 0,Y 397.378,Z 270.609,A -85,B 0,C 180,E1 -11343.04,E2 -11343.04} C_VEL
LIN {X 0,Y 397.367,Z 270.61,A -85,B 0,C 180,E1 -11347.111,E2 -11347.111} C_VEL
LIN {X 0,Y 397.221,Z 270.633,A -85,B 0,C 180,E1 -11350.19,E2 -11350.19} C_VEL
LIN {X 0,Y 397.229,Z 270.627,A -85,B 0,C 180,E1 -11353.32,E2 -11353.32} C_VEL
LIN {X 0,Y 397.183,Z 270.633,A -85,B 0,C 180,E1 -11357.154,E2 -11357.154} C_VEL
LIN {X 0,Y 397.103,Z 270.644,A -85,B 0,C 180,E1 -11360.728,E2 -11360.728} C_VEL
LIN {X 0,Y 397.133,Z 270.644,A -85,B 0,C 180,E1 -11364.017,E2 -11364.017} C_VEL
LIN {X 0,Y 397.194,Z 270.632,A -85,B 0,C 180,E1 -11367.389,E2 -11367.389} C_VEL
LIN {X 0,Y 397.077,Z 270.646,A -85,B 0,C 180,E1 -11370.881,E2 -11370.881} C_VEL
LIN {X 0,Y 397.124,Z 270.642,A -85,B 0,C 180,E1 -11374.492,E2 -11374.492} C_VEL
LIN {X 0,Y 397.104,Z 270.646,A -85,B 0,C 180,E1 -11378.273,E2 -11378.273} C_VEL
LIN {X 0,Y 397.086,Z 270.645,A -85,B 0,C 180,E1 -11380.907,E2 -11380.907} C_VEL
LIN {X 0,Y 397.101,Z 270.648,A -85,B 0,C 180,E1 -11383.646,E2 -11383.646} C_VEL
LIN {X 0,Y 397.157,Z 270.636,A -85,B 0,C 180,E1 -11386.51,E2 -11386.51} C_VEL
LIN {X 0,Y 397.118,Z 270.645,A -85,B 0,C 180,E1 -11389.549,E2 -11389.549} C_VEL
LIN {X 0,Y 397.092,Z 270.644,A -85,B 0,C 180,E1 -11392.789,E2 -11392.789} C_VEL
LIN {X 0,Y 397.112,Z 270.643,A -85,B 0,C 180,E1 -11396.281,E2 -11396.281} C_VEL
LIN {X 0,Y 397.106,Z 270.644,A -85,B 0,C 180,E1 -11400.132,E2 -11400.132} C_VEL
LIN {X 0,Y 397.187,Z 270.632,A -85,B 0,C 180,E1 -11402.609,E2 -11402.609} C_VEL
LIN {X 0,Y 397.124,Z 270.642,A -85,B 0,C 180,E1 -11405.981,E2 -11405.981} C_VEL
LIN {X 0,Y 397.129,Z 270.644,A -85,B 0,C 180,E1 -11409.703,E2 -11409.703} C_VEL
LIN {X 0,Y 397.172,Z 270.635,A -85,B 0,C 180,E1 -11412.844,E2 -11412.844} C_VEL
LIN {X 0,Y 397.216,Z 270.629,A -85,B 0,C 180,E1 -11416.678,E2 -11416.678} C_VEL
LIN {X 0,Y 397.219,Z 270.63,A -85,B 0,C 180,E1 -11419.808,E2 -11419.808} C_VEL
LIN {X 0,Y 397.351,Z 270.614,A -85,B 0,C 180,E1 -11422.887,E2 -11422.887} C_VEL
LIN {X 0,Y 397.207,Z 270.632,A -85,B 0,C 180,E1 -11424.924,E2 -11424.924} C_VEL
LIN {X 0,Y 397.227,Z 270.732,A -85,B 0,C 180,E1 -11428.986,E2 -11428.986} C_VEL
LIN {X 0,Y 396.657,Z 275.064,A -85,B 0,C 180,E1 -11434.063,E2 -11434.063} C_VEL
LIN {X 0,Y 396.576,Z 277.998,A -85,B 0,C 180,E1 -11437.337,E2 -11437.337} C_VEL
LIN {X 0,Y 399.386,Z 286.001,A -85,B 0,C 180,E1 -11437.726,E2 -11437.726} C_VEL
LIN {X 0,Y 404.558,Z 301.007,A -85,B 0,C 180,E1 -11438.597,E2 -11438.597} C_VEL
LIN {X 0,Y 407.562,Z 311.99,A -85,B 0,C 180,E1 -11439.318,E2 -11439.318} C_VEL
LIN {X 0,Y 406.445,Z 326.651,A -85,B 0,C 180,E1 -11440.145,E2 -11440.145} C_VEL
LIN {X 0,Y 405.278,Z 340.218,A -85,B 0,C 180,E1 -11441.123,E2 -11441.123} C_VEL
LIN {X 0,Y 404.105,Z 352.631,A -85,B 0,C 180,E1 -11442.22,E2 -11442.22} C_VEL
LIN {X 0,Y 402.824,Z 364.615,A -85,B 0,C 180,E1 -11443.494,E2 -11443.494} C_VEL
LIN {X 0,Y 401.495,Z 376.134,A -85,B 0,C 180,E1 -11444.962,E2 -11444.962} C_VEL
LIN {X 0,Y 400.443,Z 384.781,A -85,B 0,C 180,E1 -11446.258,E2 -11446.258} C_VEL
LIN {X 0,Y 399.346,Z 388.697,A -85,B 0,C 180,E1 -11446.871,E2 -11446.871} C_VEL
LIN {X 0,Y 395.814,Z 394.824,A -85,B 0,C 180,E1 -11447.872,E2 -11447.872} C_VEL
LIN {X 0,Y 392.329,Z 400.584,A -85,B 0,C 180,E1 -11448.939,E2 -11448.939} C_VEL
LIN {X 0,Y 391.317,Z 403.748,A -85,B 0,C 180,E1 -11449.646,E2 -11449.646} C_VEL
LIN {X 0,Y 390.427,Z 411.277,A -85,B 0,C 180,E1 -11451.654,E2 -11451.654} C_VEL
LIN {X 0,Y 389.825,Z 416.512,A -85,B 0,C 180,E1 -11453.367,E2 -11453.367} C_VEL
LIN {X 0,Y 389.325,Z 422.045,A -85,B 0,C 180,E1 -11455.673,E2 -11455.673} C_VEL
LIN {X 0,Y 388.991,Z 425.629,A -85,B 0,C 180,E1 -11457.716,E2 -11457.716} C_VEL
LIN {X 0,Y 388.735,Z 428.102,A -85,B 0,C 180,E1 -11459.8,E2 -11459.8} C_VEL
LIN {X 0,Y 388.68,Z 429.373,A -85,B 0,C 180,E1 -11461.809,E2 -11461.809} C_VEL
LIN {X 0,Y 388.645,Z 429.523,A -85,B 0,C 180,E1 -11464.095,E2 -11464.095} C_VEL
LIN {X 0,Y 388.692,Z 428.908,A -85,B 0,C 180,E1 -11465.549,E2 -11465.549} C_VEL
LIN {X 0,Y 388.858,Z 427.376,A -85,B 0,C 180,E1 -11467.326,E2 -11467.326} C_VEL
LIN {X 0,Y 389.162,Z 424.845,A -85,B 0,C 180,E1 -11469.202,E2 -11469.202} C_VEL
LIN {X 0,Y 389.554,Z 420.979,A -85,B 0,C 180,E1 -11471.243,E2 -11471.243} C_VEL
LIN {X 0,Y 390.096,Z 416.08,A -85,B 0,C 180,E1 -11473.204,E2 -11473.204} C_VEL
LIN {X 0,Y 390.763,Z 410.31,A -85,B 0,C 180,E1 -11475.032,E2 -11475.032} C_VEL
LIN {X 0,Y 391.774,Z 402.59,A -85,B 0,C 180,E1 -11477.027,E2 -11477.027} C_VEL
LIN {X 0,Y 392.823,Z 394.69,A -85,B 0,C 180,E1 -11478.712,E2 -11478.712} C_VEL
LIN {X 0,Y 394.096,Z 384.861,A -85,B 0,C 180,E1 -11480.468,E2 -11480.468} C_VEL
LIN {X 0,Y 395.493,Z 374.216,A -85,B 0,C 180,E1 -11482.049,E2 -11482.049} C_VEL
LIN {X 0,Y 396.996,Z 362.967,A -85,B 0,C 180,E1 -11483.441,E2 -11483.441} C_VEL
LIN {X 0,Y 398.376,Z 350.769,A -85,B 0,C 180,E1 -11484.709,E2 -11484.709} C_VEL
LIN {X 0,Y 399.63,Z 338.623,A -85,B 0,C 180,E1 -11485.755,E2 -11485.755} C_VEL
LIN {X 0,Y 400.917,Z 324.839,A -85,B 0,C 180,E1 -11486.71,E2 -11486.71} C_VEL
LIN {X 0,Y 401.639,Z 314.423,A -85,B 0,C 180,E1 -11487.296,E2 -11487.296} C_VEL
LIN {X 0,Y 397.337,Z 300.416,A -85,B 0,C 180,E1 -11488.292,E2 -11488.292} C_VEL
LIN {X 0,Y 392.291,Z 287.163,A -85,B 0,C 180,E1 -11489.15,E2 -11489.15} C_VEL
LIN {X 0,Y 389.802,Z 281.369,A -85,B 0,C 180,E1 -11489.494,E2 -11489.494} C_VEL
LIN {X 0,Y 389.608,Z 280.439,A -85,B 0,C 180,E1 -11489.553,E2 -11489.553} C_VEL
LIN {X 0,Y 389.725,Z 278.472,A -85,B 0,C 180,E1 -11492.081,E2 -11492.081} C_VEL
LIN {X 0,Y 389.832,Z 275.886,A -85,B 0,C 180,E1 -11495.504,E2 -11495.504} C_VEL
LIN {X 0,Y 389.97,Z 273.4,A -85,B 0,C 180,E1 -11498.874,E2 -11498.874} C_VEL
LIN {X 0,Y 389.985,Z 271.851,A -85,B 0,C 180,E1 -11501.073,E2 -11501.073} C_VEL
LIN {X 0,Y 390.116,Z 271.522,A -85,B 0,C 180,E1 -11503.249,E2 -11503.249} C_VEL
LIN {X 0,Y 390.187,Z 271.509,A -85,B 0,C 180,E1 -11506.563,E2 -11506.563} C_VEL
LIN {X 0,Y 390.199,Z 271.507,A -85,B 0,C 180,E1 -11510.672,E2 -11510.672} C_VEL
LIN {X 0,Y 390.313,Z 271.492,A -85,B 0,C 180,E1 -11512.76,E2 -11512.76} C_VEL
LIN {X 0,Y 390.223,Z 271.504,A -85,B 0,C 180,E1 -11514.835,E2 -11514.835} C_VEL
LIN {X 0,Y 390.416,Z 271.478,A -85,B 0,C 180,E1 -11517.938,E2 -11517.938} C_VEL
LIN {X 0,Y 390.545,Z 271.461,A -85,B 0,C 180,E1 -11520.001,E2 -11520.001} C_VEL
LIN {X 0,Y 390.311,Z 271.493,A -85,B 0,C 180,E1 -11523.098,E2 -11523.098} C_VEL
LIN {X 0,Y 390.326,Z 271.488,A -85,B 0,C 180,E1 -11526.203,E2 -11526.203} C_VEL
LIN {X 0,Y 390.31,Z 271.49,A -85,B 0,C 180,E1 -11528.283,E2 -11528.283} C_VEL
LIN {X 0,Y 390.167,Z 271.508,A -85,B 0,C 180,E1 -11532.484,E2 -11532.484} C_VEL
LIN {X 0,Y 390.136,Z 271.513,A -85,B 0,C 180,E1 -11535.678,E2 -11535.678} C_VEL
LIN {X 0,Y 390.103,Z 271.517,A -85,B 0,C 180,E1 -11538.923,E2 -11538.923} C_VEL
LIN {X 0,Y 390.038,Z 271.527,A -85,B 0,C 180,E1 -11542.235,E2 -11542.235} C_VEL
LIN {X 0,Y 390.117,Z 271.516,A -85,B 0,C 180,E1 -11545.744,E2 -11545.744} C_VEL
LIN {X 0,Y 390.056,Z 271.526,A -85,B 0,C 180,E1 -11549.111,E2 -11549.111} C_VEL
LIN {X 0,Y 390.041,Z 271.532,A -85,B 0,C 180,E1 -11552.723,E2 -11552.723} C_VEL
LIN {X 0,Y 390.059,Z 271.6,A -85,B 0,C 180,E1 -11556.297,E2 -11556.297} C_VEL
LIN {X 0,Y 390.74,Z 275.238,A -85,B 0,C 180,E1 -11559.34,E2 -11559.34} C_VEL
LIN {X 0,Y 391.44,Z 279.665,A -85,B 0,C 180,E1 -11562.599,E2 -11562.599} C_VEL
LIN {X 0,Y 392.364,Z 284.366,A -85,B 0,C 180,E1 -11565.765,E2 -11565.765} C_VEL
LIN {X 0,Y 392.739,Z 287.826,A -85,B 0,C 180,E1 -11567.884,E2 -11567.884} C_VEL
LIN {X 0,Y 392.398,Z 292.267,A -85,B 0,C 180,E1 -11570.368,E2 -11570.368} C_VEL
LIN {X 0,Y 391.723,Z 298.831,A -85,B 0,C 180,E1 -11573.839,E2 -11573.839} C_VEL
LIN {X 0,Y 391.119,Z 305.929,A -85,B 0,C 180,E1 -11577.381,E2 -11577.381} C_VEL
LIN {X 0,Y 390.634,Z 313.413,A -85,B 0,C 180,E1 -11580.938,E2 -11580.938} C_VEL
LIN {X 0,Y 390.29,Z 319.213,A -85,B 0,C 180,E1 -11583.513,E2 -11583.513} C_VEL
LIN {X 0,Y 394.672,Z 335.706,A -85,B 0,C 180,E1 -11584.277,E2 -11584.277} C_VEL
LIN {X 0,Y 397.892,Z 351.638,A -85,B 0,C 180,E1 -11585.154,E2 -11585.154} C_VEL
LIN {X 0,Y 400.187,Z 363.688,A -85,B 0,C 180,E1 -11585.954,E2 -11585.954} C_VEL
LIN {X 0,Y 398.963,Z 377.867,A -85,B 0,C 180,E1 -11586.84,E2 -11586.84} C_VEL
LIN {X 0,Y 397.399,Z 391.82,A -85,B 0,C 180,E1 -11587.927,E2 -11587.927} C_VEL
LIN {X 0,Y 395.836,Z 405.065,A -85,B 0,C 180,E1 -11589.201,E2 -11589.201} C_VEL
LIN {X 0,Y 394.515,Z 416.073,A -85,B 0,C 180,E1 -11590.469,E2 -11590.469} C_VEL
LIN {X 0,Y 393.184,Z 427.511,A -85,B 0,C 180,E1 -11592.042,E2 -11592.042} C_VEL
LIN {X 0,Y 391.772,Z 438.494,A -85,B 0,C 180,E1 -11593.857,E2 -11593.857} C_VEL
LIN {X 0,Y 390.707,Z 447.665,A -85,B 0,C 180,E1 -11595.681,E2 -11595.681} C_VEL
LIN {X 0,Y 389.962,Z 455.297,A -85,B 0,C 180,E1 -11597.511,E2 -11597.511} C_VEL
LIN {X 0,Y 389.494,Z 460.784,A -85,B 0,C 180,E1 -11599.079,E2 -11599.079} C_VEL
LIN {X 0,Y 389.052,Z 466.787,A -85,B 0,C 180,E1 -11601.168,E2 -11601.168} C_VEL
LIN {X 0,Y 388.913,Z 470.367,A -85,B 0,C 180,E1 -11602.734,E2 -11602.734} C_VEL
LIN {X 0,Y 388.783,Z 473.994,A -85,B 0,C 180,E1 -11604.815,E2 -11604.815} C_VEL
LIN {X 0,Y 388.708,Z 476.387,A -85,B 0,C 180,E1 -11606.891,E2 -11606.891} C_VEL
LIN {X 0,Y 388.785,Z 477.146,A -85,B 0,C 180,E1 -11607.929,E2 -11607.929} C_VEL
LIN {X 0,Y 388.674,Z 477.772,A -85,B 0,C 180,E1 -11610.001,E2 -11610.001} C_VEL
LIN {X 0,Y 388.783,Z 477.19,A -85,B 0,C 180,E1 -11612.073,E2 -11612.073} C_VEL
LIN {X 0,Y 388.683,Z 475.423,A -85,B 0,C 180,E1 -11614.148,E2 -11614.148} C_VEL
LIN {X 0,Y 388.836,Z 472.473,A -85,B 0,C 180,E1 -11616.226,E2 -11616.226} C_VEL
LIN {X 0,Y 388.978,Z 468.254,A -85,B 0,C 180,E1 -11618.312,E2 -11618.312} C_VEL
LIN {X 0,Y 389.306,Z 462.664,A -85,B 0,C 180,E1 -11620.401,E2 -11620.401} C_VEL
LIN {X 0,Y 389.993,Z 455.566,A -85,B 0,C 180,E1 -11622.49,E2 -11622.49} C_VEL
LIN {X 0,Y 390.719,Z 447.976,A -85,B 0,C 180,E1 -11624.32,E2 -11624.32} C_VEL
LIN {X 0,Y 391.798,Z 438.842,A -85,B 0,C 180,E1 -11626.144,E2 -11626.144} C_VEL
LIN {X 0,Y 393.211,Z 427.866,A -85,B 0,C 180,E1 -11627.958,E2 -11627.958} C_VEL
LIN {X 0,Y 394.536,Z 416.387,A -85,B 0,C 180,E1 -11629.538,E2 -11629.538} C_VEL
LIN {X 0,Y 396.02,Z 404.222,A -85,B 0,C 180,E1 -11630.926,E2 -11630.926} C_VEL
LIN {X 0,Y 397.514,Z 390.634,A -85,B 0,C 180,E1 -11632.205,E2 -11632.205} C_VEL
LIN {X 0,Y 399.118,Z 376.378,A -85,B 0,C 180,E1 -11633.276,E2 -11633.276} C_VEL
LIN {X 0,Y 400.155,Z 363.845,A -85,B 0,C 180,E1 -11634.035,E2 -11634.035} C_VEL
LIN {X 0,Y 397.328,Z 349.033,A -85,B 0,C 180,E1 -11634.972,E2 -11634.972} C_VEL
LIN {X 0,Y 393.861,Z 333.745,A -85,B 0,C 180,E1 -11635.771,E2 -11635.771} C_VEL
LIN {X 0,Y 390.324,Z 320.144,A -85,B 0,C 180,E1 -11636.389,E2 -11636.389} C_VEL
LIN {X 0,Y 390.906,Z 311.873,A -85,B 0,C 180,E1 -11640.226,E2 -11640.226} C_VEL
LIN {X 0,Y 391.424,Z 304.398,A -85,B 0,C 180,E1 -11643.822,E2 -11643.822} C_VEL
LIN {X 0,Y 392.038,Z 298.216,A -85,B 0,C 180,E1 -11646.91,E2 -11646.91} C_VEL
LIN {X 0,Y 392.635,Z 292.026,A -85,B 0,C 180,E1 -11650.12,E2 -11650.12} C_VEL
LIN {X 0,Y 392.802,Z 288.35,A -85,B 0,C 180,E1 -11652.118,E2 -11652.118} C_VEL
LIN {X 0,Y 392.409,Z 284.576,A -85,B 0,C 180,E1 -11654.306,E2 -11654.306} C_VEL
LIN {X 0,Y 391.493,Z 279.579,A -85,B 0,C 180,E1 -11657.395,E2 -11657.395} C_VEL
LIN {X 0,Y 390.55,Z 274.18,A -85,B 0,C 180,E1 -11660.962,E2 -11660.962} C_VEL
LIN {X 0,Y 390.064,Z 271.523,A -85,B 0,C 180,E1 -11662.968,E2 -11662.968} C_VEL
LIN {X 0,Y 390.074,Z 271.521,A -85,B 0,C 180,E1 -11666.045,E2 -11666.045} C_VEL
LIN {X 0,Y 390.052,Z 271.521,A -85,B 0,C 180,E1 -11669.869,E2 -11669.869} C_VEL
LIN {X 0,Y 390.12,Z 271.514,A -85,B 0,C 180,E1 -11673.231,E2 -11673.231} C_VEL
LIN {X 0,Y 390.113,Z 271.519,A -85,B 0,C 180,E1 -11676.75,E2 -11676.75} C_VEL
LIN {X 0,Y 390.11,Z 271.514,A -85,B 0,C 180,E1 -11679.982,E2 -11679.982} C_VEL
LIN {X 0,Y 390.144,Z 271.51,A -85,B 0,C 180,E1 -11683.248,E2 -11683.248} C_VEL
LIN {X 0,Y 390.2,Z 271.508,A -85,B 0,C 180,E1 -11686.561,E2 -11686.561} C_VEL
LIN {X 0,Y 390.209,Z 271.506,A -85,B 0,C 180,E1 -11690.67,E2 -11690.67} C_VEL
LIN {X 0,Y 390.304,Z 271.49,A -85,B 0,C 180,E1 -11693.797,E2 -11693.797} C_VEL
LIN {X 0,Y 390.423,Z 271.476,A -85,B 0,C 180,E1 -11697.936,E2 -11697.936} C_VEL
LIN {X 0,Y 390.555,Z 271.461,A -85,B 0,C 180,E1 -11699.999,E2 -11699.999} C_VEL
LIN {X 0,Y 390.312,Z 271.489,A -85,B 0,C 180,E1 -11703.095,E2 -11703.095} C_VEL
LIN {X 0,Y 390.312,Z 271.489,A -85,B 0,C 180,E1 -11706.65,E2 -11706.65} C_VEL
LIN {X 0,Y 390.208,Z 271.501,A -85,B 0,C 180,E1 -11709.327,E2 -11709.327} C_VEL
LIN {X 0,Y 390.197,Z 271.503,A -85,B 0,C 180,E1 -11713.437,E2 -11713.437} C_VEL
LIN {X 0,Y 390.15,Z 271.509,A -85,B 0,C 180,E1 -11717.306,E2 -11717.306} C_VEL
LIN {X 0,Y 390.088,Z 271.52,A -85,B 0,C 180,E1 -11720.469,E2 -11720.469} C_VEL
LIN {X 0,Y 390.09,Z 271.516,A -85,B 0,C 180,E1 -11723.349,E2 -11723.349} C_VEL
LIN {X 0,Y 390.113,Z 271.514,A -85,B 0,C 180,E1 -11726.767,E2 -11726.767} C_VEL
LIN {X 0,Y 390.038,Z 271.526,A -85,B 0,C 180,E1 -11730.298,E2 -11730.298} C_VEL
LIN {X 0,Y 390.066,Z 271.524,A -85,B 0,C 180,E1 -11734.023,E2 -11734.023} C_VEL
LIN {X 0,Y 390.043,Z 271.525,A -85,B 0,C 180,E1 -11737.55,E2 -11737.55} C_VEL
LIN {X 0,Y 390.054,Z 271.521,A -85,B 0,C 180,E1 -11740.82,E2 -11740.82} C_VEL
LIN {X 0,Y 390.057,Z 271.526,A -85,B 0,C 180,E1 -11743.886,E2 -11743.886} C_VEL
LIN {X 0,Y 390.11,Z 271.513,A -85,B 0,C 180,E1 -11746.796,E2 -11746.796} C_VEL
LIN {X 0,Y 390.072,Z 271.522,A -85,B 0,C 180,E1 -11749.562,E2 -11749.562} C_VEL
LIN {X 0,Y 390.041,Z 271.523,A -85,B 0,C 180,E1 -11752.447,E2 -11752.447} C_VEL
LIN {X 0,Y 390.061,Z 271.523,A -85,B 0,C 180,E1 -11756.044,E2 -11756.044} C_VEL
LIN {X 0,Y 390.044,Z 271.526,A -85,B 0,C 180,E1 -11759.866,E2 -11759.866} C_VEL
LIN {X 0,Y 390.105,Z 271.517,A -85,B 0,C 180,E1 -11763.231,E2 -11763.231} C_VEL
LIN {X 0,Y 390.098,Z 271.515,A -85,B 0,C 180,E1 -11766.749,E2 -11766.749} C_VEL
LIN {X 0,Y 390.095,Z 271.517,A -85,B 0,C 180,E1 -11769.982,E2 -11769.982} C_VEL
LIN {X 0,Y 390.128,Z 271.516,A -85,B 0,C 180,E1 -11773.247,E2 -11773.247} C_VEL
LIN {X 0,Y 390.185,Z 271.504,A -85,B 0,C 180,E1 -11776.56,E2 -11776.56} C_VEL
LIN {X 0,Y 390.169,Z 271.51,A -85,B 0,C 180,E1 -11779.622,E2 -11779.622} C_VEL
LIN {X 0,Y 390.306,Z 271.49,A -85,B 0,C 180,E1 -11782.758,E2 -11782.758} C_VEL
LIN {X 0,Y 390.184,Z 271.506,A -85,B 0,C 180,E1 -11784.832,E2 -11784.832} C_VEL
LIN {X 0,Y 390.194,Z 271.598,A -85,B 0,C 180,E1 -11788.967,E2 -11788.967} C_VEL
LIN {X 0,Y 389.618,Z 275.974,A -85,B 0,C 180,E1 -11794.137,E2 -11794.137} C_VEL
LIN {X 0,Y 389.522,Z 278.303,A -85,B 0,C 180,E1 -11796.844,E2 -11796.844} C_VEL
LIN {X 0,Y 391.352,Z 283.583,A -85,B 0,C 180,E1 -11797.115,E2 -11797.115} C_VEL
LIN {X 0,Y 396.574,Z 298.409,A -85,B 0,C 180,E1 -11797.969,E2 -11797.969} C_VEL
LIN {X 0,Y 400.557,Z 311.665,A -85,B 0,C 180,E1 -11798.856,E2 -11798.856} C_VEL
LIN {X 0,Y 400.924,Z 314.27,A -85,B 0,C 180,E1 -11799.019,E2 -11799.019} C_VEL
LIN {X 0,Y 399.74,Z 328.772,A -85,B 0,C 180,E1 -11799.876,E2 -11799.876} C_VEL
LIN {X 0,Y 398.473,Z 342.738,A -85,B 0,C 180,E1 -11800.929,E2 -11800.929} C_VEL
LIN {X 0,Y 397.111,Z 355.682,A -85,B 0,C 180,E1 -11802.131,E2 -11802.131} C_VEL
LIN {X 0,Y 395.649,Z 368.753,A -85,B 0,C 180,E1 -11803.612,E2 -11803.612} C_VEL
LIN {X 0,Y 394.158,Z 380.637,A -85,B 0,C 180,E1 -11805.247,E2 -11805.247} C_VEL
LIN {X 0,Y 392.946,Z 390.553,A -85,B 0,C 180,E1 -11806.895,E2 -11806.895} C_VEL
LIN {X 0,Y 391.672,Z 400.307,A -85,B 0,C 180,E1 -11808.843,E2 -11808.843} C_VEL
LIN {X 0,Y 391.317,Z 403.748,A -85,B 0,C 180,E1 -11809.646,E2 -11809.646} C_VEL
LIN {X 0,Y 390.324,Z 406.816,A -85,B 0,C 180,E1 -11810.372,E2 -11810.372} C_VEL
LIN {X 0,Y 386.94,Z 411.51,A -85,B 0,C 180,E1 -11811.56,E2 -11811.56} C_VEL
LIN {X 0,Y 383.599,Z 415.784,A -85,B 0,C 180,E1 -11812.804,E2 -11812.804} C_VEL
LIN {X 0,Y 382.694,Z 418.032,A -85,B 0,C 180,E1 -11813.608,E2 -11813.608} C_VEL
LIN {X 0,Y 382.239,Z 422.829,A -85,B 0,C 180,E1 -11815.723,E2 -11815.723} C_VEL
LIN {X 0,Y 381.863,Z 426.506,A -85,B 0,C 180,E1 -11817.946,E2 -11817.946} C_VEL
LIN {X 0,Y 381.645,Z 428.782,A -85,B 0,C 180,E1 -11820.063,E2 -11820.063} C_VEL
LIN {X 0,Y 381.575,Z 429.938,A -85,B 0,C 180,E1 -11822.284,E2 -11822.284} C_VEL
LIN {X 0,Y 381.582,Z 429.977,A -85,B 0,C 180,E1 -11824.026,E2 -11824.026} C_VEL
LIN {X 0,Y 381.657,Z 429,A -85,B 0,C 180,E1 -11826.104,E2 -11826.104} C_VEL
LIN {X 0,Y 381.849,Z 427.554,A -85,B 0,C 180,E1 -11827.684,E2 -11827.684} C_VEL
LIN {X 0,Y 382.229,Z 424.113,A -85,B 0,C 180,E1 -11830.055,E2 -11830.055} C_VEL
LIN {X 0,Y 382.701,Z 419.886,A -85,B 0,C 180,E1 -11832.089,E2 -11832.089} C_VEL
LIN {X 0,Y 383.335,Z 414.318,A -85,B 0,C 180,E1 -11834.16,E2 -11834.16} C_VEL
LIN {X 0,Y 384.173,Z 408.293,A -85,B 0,C 180,E1 -11835.962,E2 -11835.962} C_VEL
LIN {X 0,Y 385.237,Z 400.448,A -85,B 0,C 180,E1 -11837.895,E2 -11837.895} C_VEL
LIN {X 0,Y 386.551,Z 391.124,A -85,B 0,C 180,E1 -11839.783,E2 -11839.783} C_VEL
LIN {X 0,Y 387.897,Z 381.438,A -85,B 0,C 180,E1 -11841.42,E2 -11841.42} C_VEL
LIN {X 0,Y 389.506,Z 369.588,A -85,B 0,C 180,E1 -11843.079,E2 -11843.079} C_VEL
LIN {X 0,Y 391.165,Z 357.048,A -85,B 0,C 180,E1 -11844.521,E2 -11844.521} C_VEL
LIN {X 0,Y 392.615,Z 344.364,A -85,B 0,C 180,E1 -11845.727,E2 -11845.727} C_VEL
LIN {X 0,Y 393.979,Z 331.088,A -85,B 0,C 180,E1 -11846.753,E2 -11846.753} C_VEL
LIN {X 0,Y 395.157,Z 316.814,A -85,B 0,C 180,E1 -11847.63,E2 -11847.63} C_VEL
LIN {X 0,Y 391.946,Z 305.269,A -85,B 0,C 180,E1 -11848.482,E2 -11848.482} C_VEL
LIN {X 0,Y 387.046,Z 291.972,A -85,B 0,C 180,E1 -11849.405,E2 -11849.405} C_VEL
LIN {X 0,Y 382.77,Z 281.916,A -85,B 0,C 180,E1 -11850.048,E2 -11850.048} C_VEL
LIN {X 0,Y 382.587,Z 280.968,A -85,B 0,C 180,E1 -11850.091,E2 -11850.091} C_VEL
LIN {X 0,Y 382.709,Z 279.002,A -85,B 0,C 180,E1 -11852.673,E2 -11852.673} C_VEL
LIN {X 0,Y 382.83,Z 276.415,A -85,B 0,C 180,E1 -11856.181,E2 -11856.181} C_VEL
LIN {X 0,Y 383.001,Z 273.952,A -85,B 0,C 180,E1 -11859.597,E2 -11859.597} C_VEL
LIN {X 0,Y 382.951,Z 272.43,A -85,B 0,C 180,E1 -11861.822,E2 -11861.822} C_VEL
LIN {X 0,Y 383.102,Z 272.392,A -85,B 0,C 180,E1 -11865.119,E2 -11865.119} C_VEL
LIN {X 0,Y 383.091,Z 272.392,A -85,B 0,C 180,E1 -11868.359,E2 -11868.359} C_VEL
LIN {X 0,Y 383.298,Z 272.367,A -85,B 0,C 180,E1 -11871.934,E2 -11871.934} C_VEL
LIN {X 0,Y 383.195,Z 272.379,A -85,B 0,C 180,E1 -11874.74,E2 -11874.74} C_VEL
LIN {X 0,Y 383.383,Z 272.354,A -85,B 0,C 180,E1 -11877.9,E2 -11877.9} C_VEL
LIN {X 0,Y 383.515,Z 272.337,A -85,B 0,C 180,E1 -11880.001,E2 -11880.001} C_VEL
LIN {X 0,Y 383.248,Z 272.373,A -85,B 0,C 180,E1 -11883.155,E2 -11883.155} C_VEL
LIN {X 0,Y 383.284,Z 272.365,A -85,B 0,C 180,E1 -11886.317,E2 -11886.317} C_VEL
LIN {X 0,Y 383.256,Z 272.368,A -85,B 0,C 180,E1 -11888.437,E2 -11888.437} C_VEL
LIN {X 0,Y 383.095,Z 272.391,A -85,B 0,C 180,E1 -11891.643,E2 -11891.643} C_VEL
LIN {X 0,Y 383.107,Z 272.386,A -85,B 0,C 180,E1 -11894.883,E2 -11894.883} C_VEL
LIN {X 0,Y 383.086,Z 272.392,A -85,B 0,C 180,E1 -11898.173,E2 -11898.173} C_VEL
LIN {X 0,Y 382.99,Z 272.402,A -85,B 0,C 180,E1 -11901.532,E2 -11901.532} C_VEL
LIN {X 0,Y 383.05,Z 272.396,A -85,B 0,C 180,E1 -11904.961,E2 -11904.961} C_VEL
LIN {X 0,Y 383.038,Z 272.401,A -85,B 0,C 180,E1 -11908.494,E2 -11908.494} C_VEL
LIN {X 0,Y 383.007,Z 272.407,A -85,B 0,C 180,E1 -11912.151,E2 -11912.151} C_VEL
LIN {X 0,Y 383.029,Z 272.471,A -85,B 0,C 180,E1 -11915.632,E2 -11915.632} C_VEL
LIN {X 0,Y 383.605,Z 275.795,A -85,B 0,C 180,E1 -11918.53,E2 -11918.53} C_VEL
LIN {X 0,Y 384.247,Z 279.49,A -85,B 0,C 180,E1 -11921.419,E2 -11921.419} C_VEL
LIN {X 0,Y 385.303,Z 285.114,A -85,B 0,C 180,E1 -11925.347,E2 -11925.347} C_VEL
LIN {X 0,Y 385.746,Z 288.676,A -85,B 0,C 180,E1 -11927.616,E2 -11927.616} C_VEL
LIN {X 0,Y 385.387,Z 293.411,A -85,B 0,C 180,E1 -11930.338,E2 -11930.338} C_VEL
LIN {X 0,Y 384.787,Z 299.242,A -85,B 0,C 180,E1 -11933.48,E2 -11933.48} C_VEL
LIN {X 0,Y 384.265,Z 305.559,A -85,B 0,C 180,E1 -11936.724,E2 -11936.724} C_VEL
LIN {X 0,Y 383.641,Z 312.993,A -85,B 0,C 180,E1 -11940.356,E2 -11940.356} C_VEL
LIN {X 0,Y 383.296,Z 318.482,A -85,B 0,C 180,E1 -11942.955,E2 -11942.955} C_VEL
LIN {X 0,Y 385.894,Z 327.902,A -85,B 0,C 180,E1 -11943.393,E2 -11943.393} C_VEL
LIN {X 0,Y 389.422,Z 342.622,A -85,B 0,C 180,E1 -11944.168,E2 -11944.168} C_VEL
LIN {X 0,Y 392.131,Z 357.3,A -85,B 0,C 180,E1 -11945.069,E2 -11945.069} C_VEL
LIN {X 0,Y 393.528,Z 364.991,A -85,B 0,C 180,E1 -11945.618,E2 -11945.618} C_VEL
LIN {X 0,Y 392.23,Z 379.341,A -85,B 0,C 180,E1 -11946.562,E2 -11946.562} C_VEL
LIN {X 0,Y 390.601,Z 392.862,A -85,B 0,C 180,E1 -11947.661,E2 -11947.661} C_VEL
LIN {X 0,Y 388.986,Z 405.842,A -85,B 0,C 180,E1 -11948.956,E2 -11948.956} C_VEL
LIN {X 0,Y 387.482,Z 417.777,A -85,B 0,C 180,E1 -11950.396,E2 -11950.396} C_VEL
LIN {X 0,Y 386.127,Z 428.742,A -85,B 0,C 180,E1 -11951.976,E2 -11951.976} C_VEL
LIN {X 0,Y 384.862,Z 438.064,A -85,B 0,C 180,E1 -11953.559,E2 -11953.559} C_VEL
LIN {X 0,Y 383.744,Z 447.233,A -85,B 0,C 180,E1 -11955.415,E2 -11955.415} C_VEL
LIN {X 0,Y 382.926,Z 454.858,A -85,B 0,C 180,E1 -11957.278,E2 -11957.278} C_VEL
LIN {X 0,Y 382.467,Z 460.342,A -85,B 0,C 180,E1 -11958.876,E2 -11958.876} C_VEL
LIN {X 0,Y 381.969,Z 466.341,A -85,B 0,C 180,E1 -11961.003,E2 -11961.003} C_VEL
LIN {X 0,Y 381.83,Z 469.924,A -85,B 0,C 180,E1 -11962.598,E2 -11962.598} C_VEL
LIN {X 0,Y 381.71,Z 473.553,A -85,B 0,C 180,E1 -11964.719,E2 -11964.719} C_VEL
LIN {X 0,Y 381.613,Z 475.948,A -85,B 0,C 180,E1 -11966.834,E2 -11966.834} C_VEL
LIN {X 0,Y 381.701,Z 476.708,A -85,B 0,C 180,E1 -11967.89,E2 -11967.89} C_VEL
LIN {X 0,Y 381.607,Z 477.337,A -85,B 0,C 180,E1 -11970.001,E2 -11970.001} C_VEL
LIN {X 0,Y 381.698,Z 476.754,A -85,B 0,C 180,E1 -11972.111,E2 -11972.111} C_VEL
LIN {X 0,Y 381.613,Z 474.986,A -85,B 0,C 180,E1 -11974.225,E2 -11974.225} C_VEL
LIN {X 0,Y 381.766,Z 472.032,A -85,B 0,C 180,E1 -11976.342,E2 -11976.342} C_VEL
LIN {X 0,Y 381.918,Z 467.808,A -85,B 0,C 180,E1 -11978.466,E2 -11978.466} C_VEL
LIN {X 0,Y 382.263,Z 462.213,A -85,B 0,C 180,E1 -11980.595,E2 -11980.595} C_VEL
LIN {X 0,Y 382.792,Z 457.025,A -85,B 0,C 180,E1 -11982.19,E2 -11982.19} C_VEL
LIN {X 0,Y 383.484,Z 449.788,A -85,B 0,C 180,E1 -11984.054,E2 -11984.054} C_VEL
LIN {X 0,Y 384.531,Z 441.108,A -85,B 0,C 180,E1 -11985.912,E2 -11985.912} C_VEL
LIN {X 0,Y 385.88,Z 430.674,A -85,B 0,C 180,E1 -11987.763,E2 -11987.763} C_VEL
LIN {X 0,Y 387.303,Z 419.515,A -85,B 0,C 180,E1 -11989.409,E2 -11989.409} C_VEL
LIN {X 0,Y 388.851,Z 407.23,A -85,B 0,C 180,E1 -11990.914,E2 -11990.914} C_VEL
LIN {X 0,Y 390.37,Z 394.383,A -85,B 0,C 180,E1 -11992.215,E2 -11992.215} C_VEL
LIN {X 0,Y 392.031,Z 380.639,A -85,B 0,C 180,E1 -11993.34,E2 -11993.34} C_VEL
LIN {X 0,Y 393.366,Z 366.65,A -85,B 0,C 180,E1 -11994.264,E2 -11994.264} C_VEL
LIN {X 0,Y 393.353,Z 364.384,A -85,B 0,C 180,E1 -11994.405,E2 -11994.405} C_VEL
LIN {X 0,Y 390.381,Z 348.705,A -85,B 0,C 180,E1 -11995.429,E2 -11995.429} C_VEL
LIN {X 0,Y 386.923,Z 333.4,A -85,B 0,C 180,E1 -11996.252,E2 -11996.252} C_VEL
LIN {X 0,Y 383.323,Z 319.799,A -85,B 0,C 180,E1 -11996.859,E2 -11996.859} C_VEL
LIN {X 0,Y 383.908,Z 311.869,A -85,B 0,C 180,E1 -12000.637,E2 -12000.637} C_VEL
LIN {X 0,Y 384.535,Z 304.009,A -85,B 0,C 180,E1 -12004.512,E2 -12004.512} C_VEL
LIN {X 0,Y 385.123,Z 297.798,A -85,B 0,C 180,E1 -12007.687,E2 -12007.687} C_VEL
LIN {X 0,Y 385.62,Z 293.35,A -85,B 0,C 180,E1 -12010.051,E2 -12010.051} C_VEL
LIN {X 0,Y 385.805,Z 289.157,A -85,B 0,C 180,E1 -12012.378,E2 -12012.378} C_VEL
LIN {X 0,Y 385.359,Z 285.297,A -85,B 0,C 180,E1 -12014.661,E2 -12014.661} C_VEL
LIN {X 0,Y 384.247,Z 279.161,A -85,B 0,C 180,E1 -12018.583,E2 -12018.583} C_VEL
LIN {X 0,Y 383.342,Z 274.158,A -85,B 0,C 180,E1 -12022.032,E2 -12022.032} C_VEL
LIN {X 0,Y 383.023,Z 272.4,A -85,B 0,C 180,E1 -12023.335,E2 -12023.335} C_VEL
LIN {X 0,Y 383.009,Z 272.402,A -85,B 0,C 180,E1 -12026.599,E2 -12026.599} C_VEL
LIN {X 0,Y 382.998,Z 272.401,A -85,B 0,C 180,E1 -12030.3,E2 -12030.3} C_VEL
LIN {X 0,Y 383.087,Z 272.389,A -85,B 0,C 180,E1 -12034.02,E2 -12034.02} C_VEL
LIN {X 0,Y 383.014,Z 272.398,A -85,B 0,C 180,E1 -12037.335,E2 -12037.335} C_VEL
LIN {X 0,Y 383.067,Z 272.396,A -85,B 0,C 180,E1 -12040.716,E2 -12040.716} C_VEL
LIN {X 0,Y 383.086,Z 272.389,A -85,B 0,C 180,E1 -12044.026,E2 -12044.026} C_VEL
LIN {X 0,Y 383.142,Z 272.382,A -85,B 0,C 180,E1 -12047.283,E2 -12047.283} C_VEL
LIN {X 0,Y 383.156,Z 272.385,A -85,B 0,C 180,E1 -12050.497,E2 -12050.497} C_VEL
LIN {X 0,Y 383.26,Z 272.367,A -85,B 0,C 180,E1 -12053.682,E2 -12053.682} C_VEL
LIN {X 0,Y 383.39,Z 272.352,A -85,B 0,C 180,E1 -12057.898,E2 -12057.898} C_VEL
LIN {X 0,Y 383.524,Z 272.336,A -85,B 0,C 180,E1 -12059.999,E2 -12059.999} C_VEL
LIN {X 0,Y 383.249,Z 272.368,A -85,B 0,C 180,E1 -12063.152,E2 -12063.152} C_VEL
LIN {X 0,Y 383.272,Z 272.367,A -85,B 0,C 180,E1 -12066.645,E2 -12066.645} C_VEL
LIN {X 0,Y 383.263,Z 272.371,A -85,B 0,C 180,E1 -12068.434,E2 -12068.434} C_VEL
LIN {X 0,Y 383.1,Z 272.387,A -85,B 0,C 180,E1 -12071.641,E2 -12071.641} C_VEL
LIN {X 0,Y 383.112,Z 272.386,A -85,B 0,C 180,E1 -12074.88,E2 -12074.88} C_VEL
LIN {X 0,Y 383.091,Z 272.394,A -85,B 0,C 180,E1 -12078.171,E2 -12078.171} C_VEL
LIN {X 0,Y 382.994,Z 272.401,A -85,B 0,C 180,E1 -12081.529,E2 -12081.529} C_VEL
LIN {X 0,Y 383.052,Z 272.393,A -85,B 0,C 180,E1 -12084.959,E2 -12084.959} C_VEL
LIN {X 0,Y 383.016,Z 272.399,A -85,B 0,C 180,E1 -12088.493,E2 -12088.493} C_VEL
LIN {X 0,Y 383.008,Z 272.403,A -85,B 0,C 180,E1 -12092.148,E2 -12092.148} C_VEL
LIN {X 0,Y 383.016,Z 272.398,A -85,B 0,C 180,E1 -12094.666,E2 -12094.666} C_VEL
LIN {X 0,Y 382.999,Z 272.405,A -85,B 0,C 180,E1 -12097.903,E2 -12097.903} C_VEL
LIN {X 0,Y 382.981,Z 272.403,A -85,B 0,C 180,E1 -12101.346,E2 -12101.346} C_VEL
LIN {X 0,Y 383.005,Z 272.4,A -85,B 0,C 180,E1 -12104.304,E2 -12104.304} C_VEL
LIN {X 0,Y 383.07,Z 272.391,A -85,B 0,C 180,E1 -12107.248,E2 -12107.248} C_VEL
LIN {X 0,Y 383.016,Z 272.398,A -85,B 0,C 180,E1 -12110.411,E2 -12110.411} C_VEL
LIN {X 0,Y 383.02,Z 272.4,A -85,B 0,C 180,E1 -12114.043,E2 -12114.043} C_VEL
LIN {X 0,Y 382.981,Z 272.407,A -85,B 0,C 180,E1 -12117.576,E2 -12117.576} C_VEL
LIN {X 0,Y 382.99,Z 272.401,A -85,B 0,C 180,E1 -12120.299,E2 -12120.299} C_VEL
LIN {X 0,Y 383.049,Z 272.393,A -85,B 0,C 180,E1 -12122.697,E2 -12122.697} C_VEL
LIN {X 0,Y 383.025,Z 272.397,A -85,B 0,C 180,E1 -12126.191,E2 -12126.191} C_VEL
LIN {X 0,Y 383.046,Z 272.399,A -85,B 0,C 180,E1 -12129.597,E2 -12129.597} C_VEL
LIN {X 0,Y 383.095,Z 272.389,A -85,B 0,C 180,E1 -12132.93,E2 -12132.93} C_VEL
LIN {X 0,Y 383.116,Z 272.385,A -85,B 0,C 180,E1 -12136.463,E2 -12136.463} C_VEL
LIN {X 0,Y 383.131,Z 272.389,A -85,B 0,C 180,E1 -12139.429,E2 -12139.429} C_VEL
LIN {X 0,Y 383.261,Z 272.367,A -85,B 0,C 180,E1 -12142.624,E2 -12142.624} C_VEL
LIN {X 0,Y 383.16,Z 272.38,A -85,B 0,C 180,E1 -12144.737,E2 -12144.737} C_VEL
LIN {X 0,Y 383.16,Z 272.485,A -85,B 0,C 180,E1 -12148.948,E2 -12148.948} C_VEL
LIN {X 0,Y 382.579,Z 276.894,A -85,B 0,C 180,E1 -12154.213,E2 -12154.213} C_VEL
LIN {X 0,Y 382.456,Z 278.747,A -85,B 0,C 180,E1 -12156.359,E2 -12156.359} C_VEL
LIN {X 0,Y 383.433,Z 281.696,A -85,B 0,C 180,E1 -12156.505,E2 -12156.505} C_VEL
LIN {X 0,Y 388.682,Z 295.915,A -85,B 0,C 180,E1 -12157.329,E2 -12157.329} C_VEL
LIN {X 0,Y 393.271,Z 310.574,A -85,B 0,C 180,E1 -12158.316,E2 -12158.316} C_VEL
LIN {X 0,Y 394.159,Z 313.87,A -85,B 0,C 180,E1 -12158.557,E2 -12158.557} C_VEL
LIN {X 0,Y 394.252,Z 316.863,A -85,B 0,C 180,E1 -12158.735,E2 -12158.735} C_VEL
LIN {X 0,Y 393.057,Z 330.841,A -85,B 0,C 180,E1 -12159.601,E2 -12159.601} C_VEL
LIN {X 0,Y 391.682,Z 345.121,A -85,B 0,C 180,E1 -12160.728,E2 -12160.728} C_VEL
LIN {X 0,Y 390.218,Z 357.807,A -85,B 0,C 180,E1 -12161.953,E2 -12161.953} C_VEL
LIN {X 0,Y 388.867,Z 369.76,A -85,B 0,C 180,E1 -12163.358,E2 -12163.358} C_VEL
LIN {X 0,Y 387.367,Z 381.113,A -85,B 0,C 180,E1 -12164.954,E2 -12164.954} C_VEL
LIN {X 0,Y 386.062,Z 391.206,A -85,B 0,C 180,E1 -12166.661,E2 -12166.661} C_VEL
LIN {X 0,Y 384.717,Z 401.137,A -85,B 0,C 180,E1 -12168.694,E2 -12168.694} C_VEL
LIN {X 0,Y 383.918,Z 407.813,A -85,B 0,C 180,E1 -12170.353,E2 -12170.353} C_VEL
LIN {X 0,Y 383.192,Z 413.693,A -85,B 0,C 180,E1 -12172.084,E2 -12172.084} C_VEL
LIN {X 0,Y 382.694,Z 418.032,A -85,B 0,C 180,E1 -12173.608,E2 -12173.608} C_VEL
LIN {X 0,Y 381.825,Z 420.154,A -85,B 0,C 180,E1 -12174.424,E2 -12174.424} C_VEL
LIN {X 0,Y 378.673,Z 423.253,A -85,B 0,C 180,E1 -12175.762,E2 -12175.762} C_VEL
LIN {X 0,Y 376.057,Z 425.386,A -85,B 0,C 180,E1 -12176.861,E2 -12176.861} C_VEL
LIN {X 0,Y 374.891,Z 426.746,A -85,B 0,C 180,E1 -12177.725,E2 -12177.725} C_VEL
LIN {X 0,Y 374.769,Z 427.149,A -85,B 0,C 180,E1 -12178.02,E2 -12178.02} C_VEL
LIN {X 0,Y 374.537,Z 429.539,A -85,B 0,C 180,E1 -12180.439,E2 -12180.439} C_VEL
LIN {X 0,Y 374.483,Z 430.397,A -85,B 0,C 180,E1 -12182.382,E2 -12182.382} C_VEL
LIN {X 0,Y 374.502,Z 430.38,A -85,B 0,C 180,E1 -12184.342,E2 -12184.342} C_VEL
LIN {X 0,Y 374.597,Z 429.413,A -85,B 0,C 180,E1 -12186.224,E2 -12186.224} C_VEL
LIN {X 0,Y 374.854,Z 427.473,A -85,B 0,C 180,E1 -12188.221,E2 -12188.221} C_VEL
LIN {X 0,Y 375.23,Z 424.325,A -85,B 0,C 180,E1 -12190.334,E2 -12190.334} C_VEL
LIN {X 0,Y 375.719,Z 420.214,A -85,B 0,C 180,E1 -12192.329,E2 -12192.329} C_VEL
LIN {X 0,Y 376.34,Z 415.062,A -85,B 0,C 180,E1 -12194.283,E2 -12194.283} C_VEL
LIN {X 0,Y 377.39,Z 407.904,A -85,B 0,C 180,E1 -12196.448,E2 -12196.448} C_VEL
LIN {X 0,Y 378.509,Z 400.129,A -85,B 0,C 180,E1 -12198.359,E2 -12198.359} C_VEL
LIN {X 0,Y 379.827,Z 391.166,A -85,B 0,C 180,E1 -12200.185,E2 -12200.185} C_VEL
LIN {X 0,Y 381.265,Z 381.48,A -85,B 0,C 180,E1 -12201.835,E2 -12201.835} C_VEL
LIN {X 0,Y 382.902,Z 369.961,A -85,B 0,C 180,E1 -12203.468,E2 -12203.468} C_VEL
LIN {X 0,Y 384.571,Z 357.786,A -85,B 0,C 180,E1 -12204.894,E2 -12204.894} C_VEL
LIN {X 0,Y 386.008,Z 345.735,A -85,B 0,C 180,E1 -12206.071,E2 -12206.071} C_VEL
LIN {X 0,Y 387.555,Z 331.484,A -85,B 0,C 180,E1 -12207.195,E2 -12207.195} C_VEL
LIN {X 0,Y 388.607,Z 317.595,A -85,B 0,C 180,E1 -12208.077,E2 -12208.077} C_VEL
LIN {X 0,Y 384.144,Z 302.914,A -85,B 0,C 180,E1 -12209.208,E2 -12209.208} C_VEL
LIN {X 0,Y 378.367,Z 288.224,A -85,B 0,C 180,E1 -12210.247,E2 -12210.247} C_VEL
LIN {X 0,Y 375.738,Z 282.385,A -85,B 0,C 180,E1 -12210.634,E2 -12210.634} C_VEL
LIN {X 0,Y 375.581,Z 281.478,A -85,B 0,C 180,E1 -12210.698,E2 -12210.698} C_VEL
LIN {X 0,Y 375.739,Z 279.117,A -85,B 0,C 180,E1 -12213.87,E2 -12213.87} C_VEL
LIN {X 0,Y 375.855,Z 276.941,A -85,B 0,C 180,E1 -12216.881,E2 -12216.881} C_VEL
LIN {X 0,Y 375.983,Z 274.523,A -85,B 0,C 180,E1 -12220.34,E2 -12220.34} C_VEL
LIN {X 0,Y 375.985,Z 273.284,A -85,B 0,C 180,E1 -12222.599,E2 -12222.599} C_VEL
LIN {X 0,Y 376.082,Z 273.265,A -85,B 0,C 180,E1 -12226.343,E2 -12226.343} C_VEL
LIN {X 0,Y 376.113,Z 273.262,A -85,B 0,C 180,E1 -12230.32,E2 -12230.32} C_VEL
LIN {X 0,Y 376.224,Z 273.246,A -85,B 0,C 180,E1 -12232.488,E2 -12232.488} C_VEL
LIN {X 0,Y 376.167,Z 273.254,A -85,B 0,C 180,E1 -12234.641,E2 -12234.641} C_VEL
LIN {X 0,Y 376.349,Z 273.23,A -85,B 0,C 180,E1 -12237.861,E2 -12237.861} C_VEL
LIN {X 0,Y 376.484,Z 273.212,A -85,B 0,C 180,E1 -12240.001,E2 -12240.001} C_VEL
LIN {X 0,Y 376.186,Z 273.253,A -85,B 0,C 180,E1 -12243.214,E2 -12243.214} C_VEL
LIN {X 0,Y 376.243,Z 273.242,A -85,B 0,C 180,E1 -12246.436,E2 -12246.436} C_VEL
LIN {X 0,Y 376.201,Z 273.247,A -85,B 0,C 180,E1 -12248.596,E2 -12248.596} C_VEL
LIN {X 0,Y 376.047,Z 273.27,A -85,B 0,C 180,E1 -12251.864,E2 -12251.864} C_VEL
LIN {X 0,Y 376.055,Z 273.264,A -85,B 0,C 180,E1 -12255.169,E2 -12255.169} C_VEL
LIN {X 0,Y 376.021,Z 273.272,A -85,B 0,C 180,E1 -12258.527,E2 -12258.527} C_VEL
LIN {X 0,Y 375.961,Z 273.279,A -85,B 0,C 180,E1 -12261.955,E2 -12261.955} C_VEL
LIN {X 0,Y 376.004,Z 273.272,A -85,B 0,C 180,E1 -12265.462,E2 -12265.462} C_VEL
LIN {X 0,Y 375.968,Z 273.28,A -85,B 0,C 180,E1 -12269.08,E2 -12269.08} C_VEL
LIN {X 0,Y 375.947,Z 273.289,A -85,B 0,C 180,E1 -12272.83,E2 -12272.83} C_VEL
LIN {X 0,Y 376.019,Z 273.392,A -85,B 0,C 180,E1 -12274.989,E2 -12274.989} C_VEL
LIN {X 0,Y 376.667,Z 277.195,A -85,B 0,C 180,E1 -12278.405,E2 -12278.405} C_VEL
LIN {X 0,Y 377.145,Z 280.061,A -85,B 0,C 180,E1 -12280.71,E2 -12280.71} C_VEL
LIN {X 0,Y 378.212,Z 285.846,A -85,B 0,C 180,E1 -12284.921,E2 -12284.921} C_VEL
LIN {X 0,Y 378.713,Z 289.545,A -85,B 0,C 180,E1 -12287.336,E2 -12287.336} C_VEL
LIN {X 0,Y 378.548,Z 293.318,A -85,B 0,C 180,E1 -12289.57,E2 -12289.57} C_VEL
LIN {X 0,Y 377.833,Z 299.657,A -85,B 0,C 180,E1 -12293.115,E2 -12293.115} C_VEL
LIN {X 0,Y 377.279,Z 305.172,A -85,B 0,C 180,E1 -12296.025,E2 -12296.025} C_VEL
LIN {X 0,Y 376.761,Z 311.257,A -85,B 0,C 180,E1 -12299.102,E2 -12299.102} C_VEL
LIN {X 0,Y 376.288,Z 317.97,A -85,B 0,C 180,E1 -12302.375,E2 -12302.375} C_VEL
LIN {X 0,Y 377.265,Z 321.493,A -85,B 0,C 180,E1 -12302.54,E2 -12302.54} C_VEL
LIN {X 0,Y 381.57,Z 337.362,A -85,B 0,C 180,E1 -12303.374,E2 -12303.374} C_VEL
LIN {X 0,Y 384.594,Z 352.944,A -85,B 0,C 180,E1 -12304.311,E2 -12304.311} C_VEL
LIN {X 0,Y 386.915,Z 366.877,A -85,B 0,C 180,E1 -12305.307,E2 -12305.307} C_VEL
LIN {X 0,Y 385.379,Z 381.877,A -85,B 0,C 180,E1 -12306.347,E2 -12306.347} C_VEL
LIN {X 0,Y 383.607,Z 395.407,A -85,B 0,C 180,E1 -12307.516,E2 -12307.516} C_VEL
LIN {X 0,Y 381.815,Z 408.987,A -85,B 0,C 180,E1 -12308.966,E2 -12308.966} C_VEL
LIN {X 0,Y 380.136,Z 421.266,A -85,B 0,C 180,E1 -12310.563,E2 -12310.563} C_VEL
LIN {X 0,Y 378.814,Z 431.621,A -85,B 0,C 180,E1 -12312.175,E2 -12312.175} C_VEL
LIN {X 0,Y 377.435,Z 441.772,A -85,B 0,C 180,E1 -12314.06,E2 -12314.06} C_VEL
LIN {X 0,Y 376.379,Z 450.228,A -85,B 0,C 180,E1 -12315.952,E2 -12315.952} C_VEL
LIN {X 0,Y 375.616,Z 458.2,A -85,B 0,C 180,E1 -12318.123,E2 -12318.123} C_VEL
LIN {X 0,Y 375.011,Z 464.553,A -85,B 0,C 180,E1 -12320.29,E2 -12320.29} C_VEL
LIN {X 0,Y 374.732,Z 469.487,A -85,B 0,C 180,E1 -12322.457,E2 -12322.457} C_VEL
LIN {X 0,Y 374.62,Z 473.116,A -85,B 0,C 180,E1 -12324.618,E2 -12324.618} C_VEL
LIN {X 0,Y 374.521,Z 475.51,A -85,B 0,C 180,E1 -12326.774,E2 -12326.774} C_VEL
LIN {X 0,Y 374.581,Z 476.732,A -85,B 0,C 180,E1 -12328.926,E2 -12328.926} C_VEL
LIN {X 0,Y 374.581,Z 476.76,A -85,B 0,C 180,E1 -12331.076,E2 -12331.076} C_VEL
LIN {X 0,Y 374.615,Z 476.317,A -85,B 0,C 180,E1 -12332.151,E2 -12332.151} C_VEL
LIN {X 0,Y 374.545,Z 474.547,A -85,B 0,C 180,E1 -12334.305,E2 -12334.305} C_VEL
LIN {X 0,Y 374.678,Z 471.587,A -85,B 0,C 180,E1 -12336.463,E2 -12336.463} C_VEL
LIN {X 0,Y 374.835,Z 467.355,A -85,B 0,C 180,E1 -12338.627,E2 -12338.627} C_VEL
LIN {X 0,Y 375.23,Z 461.751,A -85,B 0,C 180,E1 -12340.796,E2 -12340.796} C_VEL
LIN {X 0,Y 375.761,Z 456.554,A -85,B 0,C 180,E1 -12342.421,E2 -12342.421} C_VEL
LIN {X 0,Y 376.52,Z 449.306,A -85,B 0,C 180,E1 -12344.32,E2 -12344.32} C_VEL
LIN {X 0,Y 377.615,Z 440.614,A -85,B 0,C 180,E1 -12346.212,E2 -12346.212} C_VEL
LIN {X 0,Y 379.056,Z 430.17,A -85,B 0,C 180,E1 -12348.094,E2 -12348.094} C_VEL
LIN {X 0,Y 380.429,Z 419.683,A -85,B 0,C 180,E1 -12349.676,E2 -12349.676} C_VEL
LIN {X 0,Y 381.995,Z 407.876,A -85,B 0,C 180,E1 -12351.166,E2 -12351.166} C_VEL
LIN {X 0,Y 383.571,Z 395.261,A -85,B 0,C 180,E1 -12352.488,E2 -12352.488} C_VEL
LIN {X 0,Y 385.119,Z 383.188,A -85,B 0,C 180,E1 -12353.529,E2 -12353.529} C_VEL
LIN {X 0,Y 386.589,Z 369.359,A -85,B 0,C 180,E1 -12354.498,E2 -12354.498} C_VEL
LIN {X 0,Y 386.765,Z 366.027,A -85,B 0,C 180,E1 -12354.705,E2 -12354.705} C_VEL
LIN {X 0,Y 383.913,Z 350.517,A -85,B 0,C 180,E1 -12355.769,E2 -12355.769} C_VEL
LIN {X 0,Y 380.64,Z 335.614,A -85,B 0,C 180,E1 -12356.614,E2 -12356.614} C_VEL
LIN {X 0,Y 376.319,Z 319.371,A -85,B 0,C 180,E1 -12357.393,E2 -12357.393} C_VEL
LIN {X 0,Y 376.919,Z 312.087,A -85,B 0,C 180,E1 -12360.938,E2 -12360.938} C_VEL
LIN {X 0,Y 377.488,Z 305.027,A -85,B 0,C 180,E1 -12364.491,E2 -12364.491} C_VEL
LIN {X 0,Y 378.13,Z 298.652,A -85,B 0,C 180,E1 -12367.832,E2 -12367.832} C_VEL
LIN {X 0,Y 378.664,Z 293.7,A -85,B 0,C 180,E1 -12370.512,E2 -12370.512} C_VEL
LIN {X 0,Y 378.763,Z 289.931,A -85,B 0,C 180,E1 -12372.669,E2 -12372.669} C_VEL
LIN {X 0,Y 378.263,Z 285.955,A -85,B 0,C 180,E1 -12375.086,E2 -12375.086} C_VEL
LIN {X 0,Y 377.399,Z 281.23,A -85,B 0,C 180,E1 -12378.15,E2 -12378.15} C_VEL
LIN {X 0,Y 376.433,Z 275.74,A -85,B 0,C 180,E1 -12381.967,E2 -12381.967} C_VEL
LIN {X 0,Y 376.004,Z 273.274,A -85,B 0,C 180,E1 -12383.891,E2 -12383.891} C_VEL
LIN {X 0,Y 375.955,Z 273.281,A -85,B 0,C 180,E1 -12387.27,E2 -12387.27} C_VEL
LIN {X 0,Y 375.967,Z 273.28,A -85,B 0,C 180,E1 -12390.92,E2 -12390.92} C_VEL
LIN {X 0,Y 376.013,Z 273.273,A -85,B 0,C 180,E1 -12394.539,E2 -12394.539} C_VEL
LIN {X 0,Y 375.969,Z 273.275,A -85,B 0,C 180,E1 -12398.045,E2 -12398.045} C_VEL
LIN {X 0,Y 376.015,Z 273.269,A -85,B 0,C 180,E1 -12401.473,E2 -12401.473} C_VEL
LIN {X 0,Y 376.064,Z 273.267,A -85,B 0,C 180,E1 -12404.832,E2 -12404.832} C_VEL
LIN {X 0,Y 376.055,Z 273.266,A -85,B 0,C 180,E1 -12408.136,E2 -12408.136} C_VEL
LIN {X 0,Y 376.199,Z 273.247,A -85,B 0,C 180,E1 -12411.946,E2 -12411.946} C_VEL
LIN {X 0,Y 376.164,Z 273.255,A -85,B 0,C 180,E1 -12414.639,E2 -12414.639} C_VEL
LIN {X 0,Y 376.356,Z 273.227,A -85,B 0,C 180,E1 -12417.859,E2 -12417.859} C_VEL
LIN {X 0,Y 376.493,Z 273.212,A -85,B 0,C 180,E1 -12419.999,E2 -12419.999} C_VEL
LIN {X 0,Y 376.187,Z 273.247,A -85,B 0,C 180,E1 -12423.212,E2 -12423.212} C_VEL
LIN {X 0,Y 376.237,Z 273.244,A -85,B 0,C 180,E1 -12426.636,E2 -12426.636} C_VEL
LIN {X 0,Y 376.209,Z 273.248,A -85,B 0,C 180,E1 -12428.594,E2 -12428.594} C_VEL
LIN {X 0,Y 376.052,Z 273.267,A -85,B 0,C 180,E1 -12431.862,E2 -12431.862} C_VEL
LIN {X 0,Y 376.06,Z 273.263,A -85,B 0,C 180,E1 -12435.166,E2 -12435.166} C_VEL
LIN {X 0,Y 376.025,Z 273.27,A -85,B 0,C 180,E1 -12438.524,E2 -12438.524} C_VEL
LIN {X 0,Y 375.964,Z 273.28,A -85,B 0,C 180,E1 -12441.953,E2 -12441.953} C_VEL
LIN {X 0,Y 376.006,Z 273.271,A -85,B 0,C 180,E1 -12445.459,E2 -12445.459} C_VEL
LIN {X 0,Y 375.96,Z 273.276,A -85,B 0,C 180,E1 -12449.078,E2 -12449.078} C_VEL
LIN {X 0,Y 375.949,Z 273.277,A -85,B 0,C 180,E1 -12452.827,E2 -12452.827} C_VEL
LIN {X 0,Y 375.956,Z 273.278,A -85,B 0,C 180,E1 -12455.414,E2 -12455.414} C_VEL
LIN {X 0,Y 375.973,Z 273.277,A -85,B 0,C 180,E1 -12458.269,E2 -12458.269} C_VEL
LIN {X 0,Y 375.931,Z 273.283,A -85,B 0,C 180,E1 -12461.599,E2 -12461.599} C_VEL
LIN {X 0,Y 375.976,Z 273.275,A -85,B 0,C 180,E1 -12465.259,E2 -12465.259} C_VEL
LIN {X 0,Y 375.984,Z 273.274,A -85,B 0,C 180,E1 -12468.388,E2 -12468.388} C_VEL
LIN {X 0,Y 375.962,Z 273.28,A -85,B 0,C 180,E1 -12471.91,E2 -12471.91} C_VEL
LIN {X 0,Y 375.973,Z 273.277,A -85,B 0,C 180,E1 -12475.331,E2 -12475.331} C_VEL
LIN {X 0,Y 375.953,Z 273.277,A -85,B 0,C 180,E1 -12478.437,E2 -12478.437} C_VEL
LIN {X 0,Y 375.994,Z 273.273,A -85,B 0,C 180,E1 -12482.14,E2 -12482.14} C_VEL
LIN {X 0,Y 375.998,Z 273.271,A -85,B 0,C 180,E1 -12484.538,E2 -12484.538} C_VEL
LIN {X 0,Y 375.954,Z 273.278,A -85,B 0,C 180,E1 -12488.044,E2 -12488.044} C_VEL
LIN {X 0,Y 376.015,Z 273.275,A -85,B 0,C 180,E1 -12491.473,E2 -12491.473} C_VEL
LIN {X 0,Y 376.05,Z 273.265,A -85,B 0,C 180,E1 -12494.832,E2 -12494.832} C_VEL
LIN {X 0,Y 376.049,Z 273.265,A -85,B 0,C 180,E1 -12498.136,E2 -12498.136} C_VEL
LIN {X 0,Y 376.247,Z 273.241,A -85,B 0,C 180,E1 -12501.877,E2 -12501.877} C_VEL
LIN {X 0,Y 376.136,Z 273.254,A -85,B 0,C 180,E1 -12504.639,E2 -12504.639} C_VEL
LIN {X 0,Y 376.125,Z 273.383,A -85,B 0,C 180,E1 -12508.929,E2 -12508.929} C_VEL
LIN {X 0,Y 375.541,Z 277.818,A -85,B 0,C 180,E1 -12514.292,E2 -12514.292} C_VEL
LIN {X 0,Y 375.443,Z 279.132,A -85,B 0,C 180,E1 -12515.841,E2 -12515.841} C_VEL
LIN {X 0,Y 376.496,Z 282.317,A -85,B 0,C 180,E1 -12516.01,E2 -12516.01} C_VEL
LIN {X 0,Y 381.765,Z 296.5,A -85,B 0,C 180,E1 -12516.86,E2 -12516.86} C_VEL
LIN {X 0,Y 386.243,Z 310.639,A -85,B 0,C 180,E1 -12517.837,E2 -12517.837} C_VEL
LIN {X 0,Y 387.643,Z 315.718,A -85,B 0,C 180,E1 -12518.219,E2 -12518.219} C_VEL
LIN {X 0,Y 387.275,Z 322.83,A -85,B 0,C 180,E1 -12518.645,E2 -12518.645} C_VEL
LIN {X 0,Y 386.002,Z 336.327,A -85,B 0,C 180,E1 -12519.58,E2 -12519.58} C_VEL
LIN {X 0,Y 384.487,Z 350.44,A -85,B 0,C 180,E1 -12520.798,E2 -12520.798} C_VEL
LIN {X 0,Y 383.001,Z 363.401,A -85,B 0,C 180,E1 -12522.182,E2 -12522.182} C_VEL
LIN {X 0,Y 381.461,Z 375.291,A -85,B 0,C 180,E1 -12523.716,E2 -12523.716} C_VEL
LIN {X 0,Y 379.994,Z 385.993,A -85,B 0,C 180,E1 -12525.375,E2 -12525.375} C_VEL
LIN {X 0,Y 378.733,Z 394.769,A -85,B 0,C 180,E1 -12526.993,E2 -12526.993} C_VEL
LIN {X 0,Y 377.663,Z 402.705,A -85,B 0,C 180,E1 -12528.723,E2 -12528.723} C_VEL
LIN {X 0,Y 376.668,Z 410.459,A -85,B 0,C 180,E1 -12530.762,E2 -12530.762} C_VEL
LIN {X 0,Y 375.987,Z 416.014,A -85,B 0,C 180,E1 -12532.53,E2 -12532.53} C_VEL
LIN {X 0,Y 375.311,Z 421.908,A -85,B 0,C 180,E1 -12534.918,E2 -12534.918} C_VEL
LIN {X 0,Y 375.009,Z 425.256,A -85,B 0,C 180,E1 -12536.729,E2 -12536.729} C_VEL
LIN {X 0,Y 374.769,Z 427.149,A -85,B 0,C 180,E1 -12538.02,E2 -12538.02} C_VEL
LIN {X 0,Y 374.009,Z 428.296,A -85,B 0,C 180,E1 -12538.9,E2 -12538.9} C_VEL
LIN {X 0,Y 371.048,Z 429.818,A -85,B 0,C 180,E1 -12540.337,E2 -12540.337} C_VEL
LIN {X 0,Y 368.576,Z 430.595,A -85,B 0,C 180,E1 -12541.507,E2 -12541.507} C_VEL
LIN {X 0,Y 367.501,Z 430.87,A -85,B 0,C 180,E1 -12542.417,E2 -12542.417} C_VEL
LIN {X 0,Y 367.403,Z 430.894,A -85,B 0,C 180,E1 -12542.725,E2 -12542.725} C_VEL
LIN {X 0,Y 367.426,Z 430.577,A -85,B 0,C 180,E1 -12545.017,E2 -12545.017} C_VEL
LIN {X 0,Y 367.535,Z 429.676,A -85,B 0,C 180,E1 -12546.574,E2 -12546.574} C_VEL
LIN {X 0,Y 367.927,Z 426.984,A -85,B 0,C 180,E1 -12549.075,E2 -12549.075} C_VEL
LIN {X 0,Y 368.339,Z 423.509,A -85,B 0,C 180,E1 -12551.167,E2 -12551.167} C_VEL
LIN {X 0,Y 368.95,Z 418.803,A -85,B 0,C 180,E1 -12553.294,E2 -12553.294} C_VEL
LIN {X 0,Y 369.737,Z 413.138,A -85,B 0,C 180,E1 -12555.31,E2 -12555.31} C_VEL
LIN {X 0,Y 370.788,Z 406.477,A -85,B 0,C 180,E1 -12557.237,E2 -12557.237} C_VEL
LIN {X 0,Y 371.996,Z 398.73,A -85,B 0,C 180,E1 -12559.086,E2 -12559.086} C_VEL
LIN {X 0,Y 373.39,Z 389.449,A -85,B 0,C 180,E1 -12560.932,E2 -12560.932} C_VEL
LIN {X 0,Y 375.127,Z 378.265,A -85,B 0,C 180,E1 -12562.771,E2 -12562.771} C_VEL
LIN {X 0,Y 376.751,Z 367.484,A -85,B 0,C 180,E1 -12564.237,E2 -12564.237} C_VEL
LIN {X 0,Y 378.483,Z 354.897,A -85,B 0,C 180,E1 -12565.667,E2 -12565.667} C_VEL
LIN {X 0,Y 379.985,Z 342.419,A -85,B 0,C 180,E1 -12566.835,E2 -12566.835} C_VEL
LIN {X 0,Y 381.361,Z 329.793,A -85,B 0,C 180,E1 -12567.798,E2 -12567.798} C_VEL
LIN {X 0,Y 382.256,Z 319.928,A -85,B 0,C 180,E1 -12568.425,E2 -12568.425} C_VEL
LIN {X 0,Y 378.433,Z 306.832,A -85,B 0,C 180,E1 -12569.484,E2 -12569.484} C_VEL
LIN {X 0,Y 373.331,Z 293.419,A -85,B 0,C 180,E1 -12570.504,E2 -12570.504} C_VEL
LIN {X 0,Y 368.775,Z 282.946,A -85,B 0,C 180,E1 -12571.239,E2 -12571.239} C_VEL
LIN {X 0,Y 368.607,Z 282.014,A -85,B 0,C 180,E1 -12571.287,E2 -12571.287} C_VEL
LIN {X 0,Y 368.728,Z 280.036,A -85,B 0,C 180,E1 -12574.001,E2 -12574.001} C_VEL
LIN {X 0,Y 368.86,Z 277.505,A -85,B 0,C 180,E1 -12577.602,E2 -12577.602} C_VEL
LIN {X 0,Y 368.938,Z 275.133,A -85,B 0,C 180,E1 -12581.106,E2 -12581.106} C_VEL
LIN {X 0,Y 368.945,Z 274.388,A -85,B 0,C 180,E1 -12582.256,E2 -12582.256} C_VEL
LIN {X 0,Y 369.007,Z 274.148,A -85,B 0,C 180,E1 -12585.666,E2 -12585.666} C_VEL
LIN {X 0,Y 369.016,Z 274.147,A -85,B 0,C 180,E1 -12589.022,E2 -12589.022} C_VEL
LIN {X 0,Y 369.182,Z 274.123,A -85,B 0,C 180,E1 -12592.343,E2 -12592.343} C_VEL
LIN {X 0,Y 369.14,Z 274.129,A -85,B 0,C 180,E1 -12594.539,E2 -12594.539} C_VEL
LIN {X 0,Y 369.314,Z 274.106,A -85,B 0,C 180,E1 -12597.82,E2 -12597.82} C_VEL
LIN {X 0,Y 369.454,Z 274.088,A -85,B 0,C 180,E1 -12600.001,E2 -12600.001} C_VEL
LIN {X 0,Y 369.315,Z 274.105,A -85,B 0,C 180,E1 -12602.182,E2 -12602.182} C_VEL
LIN {X 0,Y 369.205,Z 274.119,A -85,B 0,C 180,E1 -12606.559,E2 -12606.559} C_VEL
LIN {X 0,Y 369.134,Z 274.128,A -85,B 0,C 180,E1 -12608.762,E2 -12608.762} C_VEL
LIN {X 0,Y 369.002,Z 274.146,A -85,B 0,C 180,E1 -12612.094,E2 -12612.094} C_VEL
LIN {X 0,Y 368.995,Z 274.144,A -85,B 0,C 180,E1 -12615.466,E2 -12615.466} C_VEL
LIN {X 0,Y 368.979,Z 274.148,A -85,B 0,C 180,E1 -12618.894,E2 -12618.894} C_VEL
LIN {X 0,Y 368.93,Z 274.157,A -85,B 0,C 180,E1 -12622.396,E2 -12622.396} C_VEL
LIN {X 0,Y 368.998,Z 274.147,A -85,B 0,C 180,E1 -12625.981,E2 -12625.981} C_VEL
LIN {X 0,Y 368.959,Z 274.153,A -85,B 0,C 180,E1 -12628.813,E2 -12628.813} C_VEL
LIN {X 0,Y 368.896,Z 274.165,A -85,B 0,C 180,E1 -12632.239,E2 -12632.239} C_VEL
LIN {X 0,Y 368.936,Z 274.214,A -85,B 0,C 180,E1 -12634.192,E2 -12634.192} C_VEL
LIN {X 0,Y 369.523,Z 277.691,A -85,B 0,C 180,E1 -12637.49,E2 -12637.49} C_VEL
LIN {X 0,Y 370.19,Z 281.388,A -85,B 0,C 180,E1 -12640.591,E2 -12640.591} C_VEL
LIN {X 0,Y 371.112,Z 286.62,A -85,B 0,C 180,E1 -12644.484,E2 -12644.484} C_VEL
LIN {X 0,Y 371.707,Z 290.514,A -85,B 0,C 180,E1 -12647.106,E2 -12647.106} C_VEL
LIN {X 0,Y 371.615,Z 293.823,A -85,B 0,C 180,E1 -12649.156,E2 -12649.156} C_VEL
LIN {X 0,Y 370.881,Z 300.082,A -85,B 0,C 180,E1 -12652.739,E2 -12652.739} C_VEL
LIN {X 0,Y 370.257,Z 306.023,A -85,B 0,C 180,E1 -12655.949,E2 -12655.949} C_VEL
LIN {X 0,Y 369.608,Z 313.401,A -85,B 0,C 180,E1 -12659.743,E2 -12659.743} C_VEL
LIN {X 0,Y 369.309,Z 317.446,A -85,B 0,C 180,E1 -12661.766,E2 -12661.766} C_VEL
LIN {X 0,Y 370.255,Z 320.939,A -85,B 0,C 180,E1 -12661.938,E2 -12661.938} C_VEL
LIN {X 0,Y 374.538,Z 336.128,A -85,B 0,C 180,E1 -12662.771,E2 -12662.771} C_VEL
LIN {X 0,Y 377.433,Z 350.301,A -85,B 0,C 180,E1 -12663.647,E2 -12663.647} C_VEL
LIN {X 0,Y 379.97,Z 365.432,A -85,B 0,C 180,E1 -12664.744,E2 -12664.744} C_VEL
LIN {X 0,Y 380.298,Z 368.218,A -85,B 0,C 180,E1 -12664.958,E2 -12664.958} C_VEL
LIN {X 0,Y 378.843,Z 381.599,A -85,B 0,C 180,E1 -12665.914,E2 -12665.914} C_VEL
LIN {X 0,Y 377.018,Z 395.095,A -85,B 0,C 180,E1 -12667.1,E2 -12667.1} C_VEL
LIN {X 0,Y 375.154,Z 408.639,A -85,B 0,C 180,E1 -12668.574,E2 -12668.574} C_VEL
LIN {X 0,Y 373.391,Z 420.898,A -85,B 0,C 180,E1 -12670.197,E2 -12670.197} C_VEL
LIN {X 0,Y 371.987,Z 431.236,A -85,B 0,C 180,E1 -12671.837,E2 -12671.837} C_VEL
LIN {X 0,Y 370.526,Z 441.36,A -85,B 0,C 180,E1 -12673.754,E2 -12673.754} C_VEL
LIN {X 0,Y 369.4,Z 449.797,A -85,B 0,C 180,E1 -12675.681,E2 -12675.681} C_VEL
LIN {X 0,Y 368.576,Z 457.767,A -85,B 0,C 180,E1 -12677.893,E2 -12677.893} C_VEL
LIN {X 0,Y 367.952,Z 464.121,A -85,B 0,C 180,E1 -12680.102,E2 -12680.102} C_VEL
LIN {X 0,Y 367.66,Z 469.055,A -85,B 0,C 180,E1 -12682.311,E2 -12682.311} C_VEL
LIN {X 0,Y 367.533,Z 472.682,A -85,B 0,C 180,E1 -12684.514,E2 -12684.514} C_VEL
LIN {X 0,Y 367.433,Z 475.075,A -85,B 0,C 180,E1 -12686.711,E2 -12686.711} C_VEL
LIN {X 0,Y 367.519,Z 476.296,A -85,B 0,C 180,E1 -12688.905,E2 -12688.905} C_VEL
LIN {X 0,Y 367.519,Z 476.324,A -85,B 0,C 180,E1 -12691.096,E2 -12691.096} C_VEL
LIN {X 0,Y 367.423,Z 475.132,A -85,B 0,C 180,E1 -12693.29,E2 -12693.29} C_VEL
LIN {X 0,Y 367.522,Z 472.771,A -85,B 0,C 180,E1 -12695.487,E2 -12695.487} C_VEL
LIN {X 0,Y 367.661,Z 469.179,A -85,B 0,C 180,E1 -12697.69,E2 -12697.69} C_VEL
LIN {X 0,Y 367.952,Z 464.269,A -85,B 0,C 180,E1 -12699.899,E2 -12699.899} C_VEL
LIN {X 0,Y 368.577,Z 457.923,A -85,B 0,C 180,E1 -12702.108,E2 -12702.108} C_VEL
LIN {X 0,Y 369.403,Z 449.955,A -85,B 0,C 180,E1 -12704.32,E2 -12704.32} C_VEL
LIN {X 0,Y 370.54,Z 441.493,A -85,B 0,C 180,E1 -12706.247,E2 -12706.247} C_VEL
LIN {X 0,Y 371.98,Z 431.31,A -85,B 0,C 180,E1 -12708.165,E2 -12708.165} C_VEL
LIN {X 0,Y 373.4,Z 420.928,A -85,B 0,C 180,E1 -12709.804,E2 -12709.804} C_VEL
LIN {X 0,Y 375.144,Z 408.522,A -85,B 0,C 180,E1 -12711.428,E2 -12711.428} C_VEL
LIN {X 0,Y 376.799,Z 396.126,A -85,B 0,C 180,E1 -12712.77,E2 -12712.77} C_VEL
LIN {X 0,Y 378.58,Z 382.608,A -85,B 0,C 180,E1 -12713.96,E2 -12713.96} C_VEL
LIN {X 0,Y 380.057,Z 368.728,A -85,B 0,C 180,E1 -12714.948,E2 -12714.948} C_VEL
LIN {X 0,Y 379.753,Z 365.306,A -85,B 0,C 180,E1 -12715.193,E2 -12715.193} C_VEL
LIN {X 0,Y 376.918,Z 349.544,A -85,B 0,C 180,E1 -12716.286,E2 -12716.286} C_VEL
LIN {X 0,Y 373.336,Z 333.787,A -85,B 0,C 180,E1 -12717.199,E2 -12717.199} C_VEL
LIN {X 0,Y 369.326,Z 318.952,A -85,B 0,C 180,E1 -12717.93,E2 -12717.93} C_VEL
LIN {X 0,Y 369.895,Z 312.335,A -85,B 0,C 180,E1 -12721.239,E2 -12721.239} C_VEL
LIN {X 0,Y 370.477,Z 305.629,A -85,B 0,C 180,E1 -12724.688,E2 -12724.688} C_VEL
LIN {X 0,Y 371.137,Z 299.461,A -85,B 0,C 180,E1 -12727.984,E2 -12727.984} C_VEL
LIN {X 0,Y 371.698,Z 294.285,A -85,B 0,C 180,E1 -12730.859,E2 -12730.859} C_VEL
LIN {X 0,Y 371.751,Z 290.809,A -85,B 0,C 180,E1 -12732.89,E2 -12732.89} C_VEL
LIN {X 0,Y 371.152,Z 286.591,A -85,B 0,C 180,E1 -12735.522,E2 -12735.522} C_VEL
LIN {X 0,Y 370.364,Z 282.274,A -85,B 0,C 180,E1 -12738.381,E2 -12738.381} C_VEL
LIN {X 0,Y 369.342,Z 276.526,A -85,B 0,C 180,E1 -12742.488,E2 -12742.488} C_VEL
LIN {X 0,Y 368.957,Z 274.152,A -85,B 0,C 180,E1 -12744.293,E2 -12744.293} C_VEL
LIN {X 0,Y 368.904,Z 274.16,A -85,B 0,C 180,E1 -12747.762,E2 -12747.762} C_VEL
LIN {X 0,Y 368.969,Z 274.147,A -85,B 0,C 180,E1 -12751.562,E2 -12751.562} C_VEL
LIN {X 0,Y 369.006,Z 274.142,A -85,B 0,C 180,E1 -12754.019,E2 -12754.019} C_VEL
LIN {X 0,Y 368.938,Z 274.15,A -85,B 0,C 180,E1 -12757.604,E2 -12757.604} C_VEL
LIN {X 0,Y 368.964,Z 274.149,A -85,B 0,C 180,E1 -12761.105,E2 -12761.105} C_VEL
LIN {X 0,Y 369.004,Z 274.148,A -85,B 0,C 180,E1 -12764.534,E2 -12764.534} C_VEL
LIN {X 0,Y 369.01,Z 274.142,A -85,B 0,C 180,E1 -12767.906,E2 -12767.906} C_VEL
LIN {X 0,Y 369.098,Z 274.131,A -85,B 0,C 180,E1 -12771.237,E2 -12771.237} C_VEL
LIN {X 0,Y 369.136,Z 274.132,A -85,B 0,C 180,E1 -12774.536,E2 -12774.536} C_VEL
LIN {X 0,Y 369.321,Z 274.103,A -85,B 0,C 180,E1 -12777.818,E2 -12777.818} C_VEL
LIN {X 0,Y 369.463,Z 274.087,A -85,B 0,C 180,E1 -12779.999,E2 -12779.999} C_VEL
LIN {X 0,Y 369.32,Z 274.107,A -85,B 0,C 180,E1 -12782.18,E2 -12782.18} C_VEL
LIN {X 0,Y 369.207,Z 274.12,A -85,B 0,C 180,E1 -12786.624,E2 -12786.624} C_VEL
LIN {X 0,Y 369.141,Z 274.127,A -85,B 0,C 180,E1 -12788.76,E2 -12788.76} C_VEL
LIN {X 0,Y 369.008,Z 274.146,A -85,B 0,C 180,E1 -12792.092,E2 -12792.092} C_VEL
LIN {X 0,Y 369,Z 274.143,A -85,B 0,C 180,E1 -12795.463,E2 -12795.463} C_VEL
LIN {X 0,Y 368.984,Z 274.145,A -85,B 0,C 180,E1 -12798.891,E2 -12798.891} C_VEL
LIN {X 0,Y 368.933,Z 274.154,A -85,B 0,C 180,E1 -12802.393,E2 -12802.393} C_VEL
LIN {X 0,Y 369,Z 274.148,A -85,B 0,C 180,E1 -12805.979,E2 -12805.979} C_VEL
LIN {X 0,Y 368.913,Z 274.156,A -85,B 0,C 180,E1 -12809.689,E2 -12809.689} C_VEL
LIN {X 0,Y 368.897,Z 274.155,A -85,B 0,C 180,E1 -12813.042,E2 -12813.042} C_VEL
LIN {X 0,Y 368.916,Z 274.157,A -85,B 0,C 180,E1 -12816.195,E2 -12816.195} C_VEL
LIN {X 0,Y 368.901,Z 274.155,A -85,B 0,C 180,E1 -12818.951,E2 -12818.951} C_VEL
LIN {X 0,Y 368.878,Z 274.163,A -85,B 0,C 180,E1 -12822.008,E2 -12822.008} C_VEL
LIN {X 0,Y 368.951,Z 274.149,A -85,B 0,C 180,E1 -12825.186,E2 -12825.186} C_VEL
LIN {X 0,Y 368.941,Z 274.152,A -85,B 0,C 180,E1 -12828.185,E2 -12828.185} C_VEL
LIN {X 0,Y 368.907,Z 274.156,A -85,B 0,C 180,E1 -12831.357,E2 -12831.357} C_VEL
LIN {X 0,Y 368.93,Z 274.152,A -85,B 0,C 180,E1 -12835.145,E2 -12835.145} C_VEL
LIN {X 0,Y 368.922,Z 274.153,A -85,B 0,C 180,E1 -12839.045,E2 -12839.045} C_VEL
LIN {X 0,Y 368.979,Z 274.151,A -85,B 0,C 180,E1 -12841.563,E2 -12841.563} C_VEL
LIN {X 0,Y 368.949,Z 274.152,A -85,B 0,C 180,E1 -12845.223,E2 -12845.223} C_VEL
LIN {X 0,Y 368.929,Z 274.153,A -85,B 0,C 180,E1 -12848.972,E2 -12848.972} C_VEL
LIN {X 0,Y 368.981,Z 274.145,A -85,B 0,C 180,E1 -12852.256,E2 -12852.256} C_VEL
LIN {X 0,Y 369.028,Z 274.139,A -85,B 0,C 180,E1 -12856.226,E2 -12856.226} C_VEL
LIN {X 0,Y 369.062,Z 274.135,A -85,B 0,C 180,E1 -12860.131,E2 -12860.131} C_VEL
LIN {X 0,Y 369.176,Z 274.12,A -85,B 0,C 180,E1 -12862.341,E2 -12862.341} C_VEL
LIN {X 0,Y 369.112,Z 274.129,A -85,B 0,C 180,E1 -12864.536,E2 -12864.536} C_VEL
LIN {X 0,Y 369.089,Z 274.284,A -85,B 0,C 180,E1 -12868.908,E2 -12868.908} C_VEL
LIN {X 0,Y 368.455,Z 279.222,A -85,B 0,C 180,E1 -12874.923,E2 -12874.923} C_VEL
LIN {X 0,Y 368.447,Z 279.538,A -85,B 0,C 180,E1 -12875.301,E2 -12875.301} C_VEL
LIN {X 0,Y 370.369,Z 285.058,A -85,B 0,C 180,E1 -12875.614,E2 -12875.614} C_VEL
LIN {X 0,Y 375.418,Z 298.594,A -85,B 0,C 180,E1 -12876.481,E2 -12876.481} C_VEL
LIN {X 0,Y 380.096,Z 313.755,A -85,B 0,C 180,E1 -12877.581,E2 -12877.581} C_VEL
LIN {X 0,Y 381.199,Z 318.452,A -85,B 0,C 180,E1 -12877.941,E2 -12877.941} C_VEL
LIN {X 0,Y 380.004,Z 331.475,A -85,B 0,C 180,E1 -12878.776,E2 -12878.776} C_VEL
LIN {X 0,Y 378.562,Z 345.529,A -85,B 0,C 180,E1 -12879.914,E2 -12879.914} C_VEL
LIN {X 0,Y 377.02,Z 358.029,A -85,B 0,C 180,E1 -12881.15,E2 -12881.15} C_VEL
LIN {X 0,Y 375.388,Z 370.894,A -85,B 0,C 180,E1 -12882.707,E2 -12882.707} C_VEL
LIN {X 0,Y 373.718,Z 382.621,A -85,B 0,C 180,E1 -12884.428,E2 -12884.428} C_VEL
LIN {X 0,Y 372.391,Z 392.038,A -85,B 0,C 180,E1 -12886.082,E2 -12886.082} C_VEL
LIN {X 0,Y 370.935,Z 401.632,A -85,B 0,C 180,E1 -12888.103,E2 -12888.103} C_VEL
LIN {X 0,Y 369.809,Z 410.049,A -85,B 0,C 180,E1 -12890.293,E2 -12890.293} C_VEL
LIN {X 0,Y 368.961,Z 416.571,A -85,B 0,C 180,E1 -12892.392,E2 -12892.392} C_VEL
LIN {X 0,Y 368.433,Z 421.111,A -85,B 0,C 180,E1 -12894.227,E2 -12894.227} C_VEL
LIN {X 0,Y 368.034,Z 424.948,A -85,B 0,C 180,E1 -12896.171,E2 -12896.171} C_VEL
LIN {X 0,Y 367.614,Z 428.316,A -85,B 0,C 180,E1 -12898.55,E2 -12898.55} C_VEL
LIN {X 0,Y 367.416,Z 430.378,A -85,B 0,C 180,E1 -12901.094,E2 -12901.094} C_VEL
LIN {X 0,Y 367.403,Z 430.894,A -85,B 0,C 180,E1 -12902.725,E2 -12902.725} C_VEL
LIN {X 0,Y 366.713,Z 430.971,A -85,B 0,C 180,E1 -12903.642,E2 -12903.642} C_VEL
LIN {X 0,Y 363.885,Z 430.766,A -85,B 0,C 180,E1 -12905.133,E2 -12905.133} C_VEL
LIN {X 0,Y 361.556,Z 430.279,A -85,B 0,C 180,E1 -12906.335,E2 -12906.335} C_VEL
LIN {X 0,Y 360.618,Z 429.611,A -85,B 0,C 180,E1 -12907.259,E2 -12907.259} C_VEL
LIN {X 0,Y 360.574,Z 429.284,A -85,B 0,C 180,E1 -12907.57,E2 -12907.57} C_VEL
LIN {X 0,Y 360.793,Z 427.927,A -85,B 0,C 180,E1 -12908.818,E2 -12908.818} C_VEL
LIN {X 0,Y 361.147,Z 425.276,A -85,B 0,C 180,E1 -12910.631,E2 -12910.631} C_VEL
LIN {X 0,Y 361.76,Z 420.887,A -85,B 0,C 180,E1 -12912.839,E2 -12912.839} C_VEL
LIN {X 0,Y 362.556,Z 415.204,A -85,B 0,C 180,E1 -12915.034,E2 -12915.034} C_VEL
LIN {X 0,Y 363.722,Z 407.986,A -85,B 0,C 180,E1 -12917.243,E2 -12917.243} C_VEL
LIN {X 0,Y 365.107,Z 399.674,A -85,B 0,C 180,E1 -12919.301,E2 -12919.301} C_VEL
LIN {X 0,Y 366.538,Z 390.608,A -85,B 0,C 180,E1 -12921.161,E2 -12921.161} C_VEL
LIN {X 0,Y 368.287,Z 380.075,A -85,B 0,C 180,E1 -12922.952,E2 -12922.952} C_VEL
LIN {X 0,Y 369.956,Z 369.443,A -85,B 0,C 180,E1 -12924.461,E2 -12924.461} C_VEL
LIN {X 0,Y 371.854,Z 356.543,A -85,B 0,C 180,E1 -12925.979,E2 -12925.979} C_VEL
LIN {X 0,Y 373.495,Z 343.556,A -85,B 0,C 180,E1 -12927.234,E2 -12927.234} C_VEL
LIN {X 0,Y 375.031,Z 330.085,A -85,B 0,C 180,E1 -12928.282,E2 -12928.282} C_VEL
LIN {X 0,Y 375.821,Z 321.536,A -85,B 0,C 180,E1 -12928.839,E2 -12928.839} C_VEL
LIN {X 0,Y 371.828,Z 307.958,A -85,B 0,C 180,E1 -12929.992,E2 -12929.992} C_VEL
LIN {X 0,Y 366.442,Z 293.987,A -85,B 0,C 180,E1 -12931.101,E2 -12931.101} C_VEL
LIN {X 0,Y 361.742,Z 283.256,A -85,B 0,C 180,E1 -12931.894,E2 -12931.894} C_VEL
LIN {X 0,Y 361.603,Z 282.532,A -85,B 0,C 180,E1 -12931.961,E2 -12931.961} C_VEL
LIN {X 0,Y 361.706,Z 280.584,A -85,B 0,C 180,E1 -12934.695,E2 -12934.695} C_VEL
LIN {X 0,Y 361.852,Z 278.079,A -85,B 0,C 180,E1 -12938.346,E2 -12938.346} C_VEL
LIN {X 0,Y 361.936,Z 275.646,A -85,B 0,C 180,E1 -12942.074,E2 -12942.074} C_VEL
LIN {X 0,Y 361.896,Z 275.039,A -85,B 0,C 180,E1 -12943.066,E2 -12943.066} C_VEL
LIN {X 0,Y 361.992,Z 275.021,A -85,B 0,C 180,E1 -12946.529,E2 -12946.529} C_VEL
LIN {X 0,Y 362.025,Z 275.016,A -85,B 0,C 180,E1 -12949.939,E2 -12949.939} C_VEL
LIN {X 0,Y 362.145,Z 275,A -85,B 0,C 180,E1 -12952.194,E2 -12952.194} C_VEL
LIN {X 0,Y 362.114,Z 275.004,A -85,B 0,C 180,E1 -12954.432,E2 -12954.432} C_VEL
LIN {X 0,Y 362.278,Z 274.982,A -85,B 0,C 180,E1 -12957.778,E2 -12957.778} C_VEL
LIN {X 0,Y 362.423,Z 274.964,A -85,B 0,C 180,E1 -12960.001,E2 -12960.001} C_VEL
LIN {X 0,Y 362.279,Z 274.982,A -85,B 0,C 180,E1 -12962.225,E2 -12962.225} C_VEL
LIN {X 0,Y 362.168,Z 274.996,A -85,B 0,C 180,E1 -12966.687,E2 -12966.687} C_VEL
LIN {X 0,Y 362.07,Z 275.008,A -85,B 0,C 180,E1 -12968.934,E2 -12968.934} C_VEL
LIN {X 0,Y 361.957,Z 275.022,A -85,B 0,C 180,E1 -12972.333,E2 -12972.333} C_VEL
LIN {X 0,Y 361.959,Z 275.021,A -85,B 0,C 180,E1 -12974.622,E2 -12974.622} C_VEL
LIN {X 0,Y 361.957,Z 275.023,A -85,B 0,C 180,E1 -12978.1,E2 -12978.1} C_VEL
LIN {X 0,Y 361.889,Z 275.03,A -85,B 0,C 180,E1 -12981.654,E2 -12981.654} C_VEL
LIN {X 0,Y 361.926,Z 275.026,A -85,B 0,C 180,E1 -12985.291,E2 -12985.291} C_VEL
LIN {X 0,Y 361.916,Z 275.03,A -85,B 0,C 180,E1 -12987.779,E2 -12987.779} C_VEL
LIN {X 0,Y 361.845,Z 275.044,A -85,B 0,C 180,E1 -12991.286,E2 -12991.286} C_VEL
LIN {X 0,Y 361.853,Z 275.052,A -85,B 0,C 180,E1 -12993.37,E2 -12993.37} C_VEL
LIN {X 0,Y 362.273,Z 277.215,A -85,B 0,C 180,E1 -12995.592,E2 -12995.592} C_VEL
LIN {X 0,Y 362.96,Z 281.248,A -85,B 0,C 180,E1 -12999.24,E2 -12999.24} C_VEL
LIN {X 0,Y 363.694,Z 285.668,A -85,B 0,C 180,E1 -13002.752,E2 -13002.752} C_VEL
LIN {X 0,Y 364.547,Z 290.238,A -85,B 0,C 180,E1 -13006.051,E2 -13006.051} C_VEL
LIN {X 0,Y 364.762,Z 292.586,A -85,B 0,C 180,E1 -13007.597,E2 -13007.597} C_VEL
LIN {X 0,Y 364.474,Z 296.086,A -85,B 0,C 180,E1 -13009.763,E2 -13009.763} C_VEL
LIN {X 0,Y 363.773,Z 302.039,A -85,B 0,C 180,E1 -13013.209,E2 -13013.209} C_VEL
LIN {X 0,Y 363.18,Z 307.711,A -85,B 0,C 180,E1 -13016.317,E2 -13016.317} C_VEL
LIN {X 0,Y 362.497,Z 315.321,A -85,B 0,C 180,E1 -13020.306,E2 -13020.306} C_VEL
LIN {X 0,Y 362.356,Z 316.924,A -85,B 0,C 180,E1 -13021.125,E2 -13021.125} C_VEL
LIN {X 0,Y 363.334,Z 320.469,A -85,B 0,C 180,E1 -13021.308,E2 -13021.308} C_VEL
LIN {X 0,Y 367.627,Z 335.319,A -85,B 0,C 180,E1 -13022.17,E2 -13022.17} C_VEL
LIN {X 0,Y 370.613,Z 349.396,A -85,B 0,C 180,E1 -13023.072,E2 -13023.072} C_VEL
LIN {X 0,Y 373.019,Z 364.643,A -85,B 0,C 180,E1 -13024.191,E2 -13024.191} C_VEL
LIN {X 0,Y 373.684,Z 368.599,A -85,B 0,C 180,E1 -13024.523,E2 -13024.523} C_VEL
LIN {X 0,Y 372.123,Z 382.943,A -85,B 0,C 180,E1 -13025.599,E2 -13025.599} C_VEL
LIN {X 0,Y 370.241,Z 396.092,A -85,B 0,C 180,E1 -13026.805,E2 -13026.805} C_VEL
LIN {X 0,Y 368.321,Z 409.369,A -85,B 0,C 180,E1 -13028.304,E2 -13028.304} C_VEL
LIN {X 0,Y 366.659,Z 420.53,A -85,B 0,C 180,E1 -13029.818,E2 -13029.818} C_VEL
LIN {X 0,Y 365.166,Z 430.857,A -85,B 0,C 180,E1 -13031.485,E2 -13031.485} C_VEL
LIN {X 0,Y 363.627,Z 440.969,A -85,B 0,C 180,E1 -13033.437,E2 -13033.437} C_VEL
LIN {X 0,Y 362.459,Z 449.4,A -85,B 0,C 180,E1 -13035.401,E2 -13035.401} C_VEL
LIN {X 0,Y 361.689,Z 455.489,A -85,B 0,C 180,E1 -13037.089,E2 -13037.089} C_VEL
LIN {X 0,Y 361.014,Z 462.224,A -85,B 0,C 180,E1 -13039.343,E2 -13039.343} C_VEL
LIN {X 0,Y 360.639,Z 467.515,A -85,B 0,C 180,E1 -13041.597,E2 -13041.597} C_VEL
LIN {X 0,Y 360.505,Z 471.497,A -85,B 0,C 180,E1 -13043.85,E2 -13043.85} C_VEL
LIN {X 0,Y 360.414,Z 473.596,A -85,B 0,C 180,E1 -13045.527,E2 -13045.527} C_VEL
LIN {X 0,Y 360.426,Z 475.397,A -85,B 0,C 180,E1 -13047.766,E2 -13047.766} C_VEL
LIN {X 0,Y 360.418,Z 476.028,A -85,B 0,C 180,E1 -13050.001,E2 -13050.001} C_VEL
LIN {X 0,Y 360.422,Z 475.436,A -85,B 0,C 180,E1 -13052.236,E2 -13052.236} C_VEL
LIN {X 0,Y 360.41,Z 473.658,A -85,B 0,C 180,E1 -13054.474,E2 -13054.474} C_VEL
LIN {X 0,Y 360.5,Z 470.681,A -85,B 0,C 180,E1 -13056.718,E2 -13056.718} C_VEL
LIN {X 0,Y 360.693,Z 466.434,A -85,B 0,C 180,E1 -13058.968,E2 -13058.968} C_VEL
LIN {X 0,Y 361.192,Z 460.817,A -85,B 0,C 180,E1 -13061.221,E2 -13061.221} C_VEL
LIN {X 0,Y 361.9,Z 453.673,A -85,B 0,C 180,E1 -13063.477,E2 -13063.477} C_VEL
LIN {X 0,Y 363.084,Z 444.807,A -85,B 0,C 180,E1 -13065.724,E2 -13065.724} C_VEL
LIN {X 0,Y 364.408,Z 435.376,A -85,B 0,C 180,E1 -13067.684,E2 -13067.684} C_VEL
LIN {X 0,Y 365.984,Z 424.905,A -85,B 0,C 180,E1 -13069.491,E2 -13069.491} C_VEL
LIN {X 0,Y 367.641,Z 413.37,A -85,B 0,C 180,E1 -13071.152,E2 -13071.152} C_VEL
LIN {X 0,Y 369.504,Z 400.709,A -85,B 0,C 180,E1 -13072.654,E2 -13072.654} C_VEL
LIN {X 0,Y 371.179,Z 388.284,A -85,B 0,C 180,E1 -13073.874,E2 -13073.874} C_VEL
LIN {X 0,Y 372.935,Z 374.086,A -85,B 0,C 180,E1 -13075,E2 -13075} C_VEL
LIN {X 0,Y 373.42,Z 368.412,A -85,B 0,C 180,E1 -13075.391,E2 -13075.391} C_VEL
LIN {X 0,Y 370.678,Z 352.658,A -85,B 0,C 180,E1 -13076.564,E2 -13076.564} C_VEL
LIN {X 0,Y 367.56,Z 337.992,A -85,B 0,C 180,E1 -13077.477,E2 -13077.477} C_VEL
LIN {X 0,Y 363.389,Z 322.626,A -85,B 0,C 180,E1 -13078.289,E2 -13078.289} C_VEL
LIN {X 0,Y 362.346,Z 318.535,A -85,B 0,C 180,E1 -13078.499,E2 -13078.499} C_VEL
LIN {X 0,Y 362.883,Z 312.561,A -85,B 0,C 180,E1 -13081.552,E2 -13081.552} C_VEL
LIN {X 0,Y 363.617,Z 305.189,A -85,B 0,C 180,E1 -13085.44,E2 -13085.44} C_VEL
LIN {X 0,Y 364.309,Z 299.041,A -85,B 0,C 180,E1 -13088.828,E2 -13088.828} C_VEL
LIN {X 0,Y 364.73,Z 294.73,A -85,B 0,C 180,E1 -13091.279,E2 -13091.279} C_VEL
LIN {X 0,Y 364.757,Z 291.992,A -85,B 0,C 180,E1 -13092.931,E2 -13092.931} C_VEL
LIN {X 0,Y 364.163,Z 287.84,A -85,B 0,C 180,E1 -13095.567,E2 -13095.567} C_VEL
LIN {X 0,Y 363.237,Z 282.806,A -85,B 0,C 180,E1 -13098.99,E2 -13098.99} C_VEL
LIN {X 0,Y 362.296,Z 277.286,A -85,B 0,C 180,E1 -13103.032,E2 -13103.032} C_VEL
LIN {X 0,Y 361.895,Z 275.034,A -85,B 0,C 180,E1 -13104.914,E2 -13104.914} C_VEL
LIN {X 0,Y 361.853,Z 275.038,A -85,B 0,C 180,E1 -13108.714,E2 -13108.714} C_VEL
LIN {X 0,Y 361.914,Z 275.026,A -85,B 0,C 180,E1 -13112.221,E2 -13112.221} C_VEL
LIN {X 0,Y 361.935,Z 275.028,A -85,B 0,C 180,E1 -13114.709,E2 -13114.709} C_VEL
LIN {X 0,Y 361.898,Z 275.03,A -85,B 0,C 180,E1 -13118.346,E2 -13118.346} C_VEL
LIN {X 0,Y 361.973,Z 275.019,A -85,B 0,C 180,E1 -13122.061,E2 -13122.061} C_VEL
LIN {X 0,Y 362.004,Z 275.015,A -85,B 0,C 180,E1 -13126.1,E2 -13126.1} C_VEL
LIN {X 0,Y 362.036,Z 275.011,A -85,B 0,C 180,E1 -13129.937,E2 -13129.937} C_VEL
LIN {X 0,Y 362.14,Z 274.997,A -85,B 0,C 180,E1 -13133.312,E2 -13133.312} C_VEL
LIN {X 0,Y 362.285,Z 274.979,A -85,B 0,C 180,E1 -13137.775,E2 -13137.775} C_VEL
LIN {X 0,Y 362.433,Z 274.962,A -85,B 0,C 180,E1 -13139.999,E2 -13139.999} C_VEL
LIN {X 0,Y 362.284,Z 274.983,A -85,B 0,C 180,E1 -13142.222,E2 -13142.222} C_VEL
LIN {X 0,Y 362.175,Z 274.995,A -85,B 0,C 180,E1 -13146.685,E2 -13146.685} C_VEL
LIN {X 0,Y 362.077,Z 275.005,A -85,B 0,C 180,E1 -13148.932,E2 -13148.932} C_VEL
LIN {X 0,Y 361.963,Z 275.024,A -85,B 0,C 180,E1 -13152.331,E2 -13152.331} C_VEL
LIN {X 0,Y 361.964,Z 275.021,A -85,B 0,C 180,E1 -13154.619,E2 -13154.619} C_VEL
LIN {X 0,Y 361.961,Z 275.025,A -85,B 0,C 180,E1 -13158.098,E2 -13158.098} C_VEL
LIN {X 0,Y 361.893,Z 275.029,A -85,B 0,C 180,E1 -13161.651,E2 -13161.651} C_VEL
LIN {X 0,Y 361.928,Z 275.023,A -85,B 0,C 180,E1 -13165.288,E2 -13165.288} C_VEL
LIN {X 0,Y 361.908,Z 275.029,A -85,B 0,C 180,E1 -13167.777,E2 -13167.777} C_VEL
LIN {X 0,Y 361.836,Z 275.037,A -85,B 0,C 180,E1 -13171.628,E2 -13171.628} C_VEL
LIN {X 0,Y 361.872,Z 275.031,A -85,B 0,C 180,E1 -13175.343,E2 -13175.343} C_VEL
LIN {X 0,Y 361.868,Z 275.031,A -85,B 0,C 180,E1 -13179.025,E2 -13179.025} C_VEL
LIN {X 0,Y 361.835,Z 275.035,A -85,B 0,C 180,E1 -13182.827,E2 -13182.827} C_VEL
LIN {X 0,Y 361.908,Z 275.031,A -85,B 0,C 180,E1 -13185.929,E2 -13185.929} C_VEL
LIN {X 0,Y 361.901,Z 275.028,A -85,B 0,C 180,E1 -13189.23,E2 -13189.23} C_VEL
LIN {X 0,Y 361.863,Z 275.032,A -85,B 0,C 180,E1 -13192.981,E2 -13192.981} C_VEL
LIN {X 0,Y 361.852,Z 275.033,A -85,B 0,C 180,E1 -13196.629,E2 -13196.629} C_VEL
LIN {X 0,Y 361.869,Z 275.037,A -85,B 0,C 180,E1 -13199.671,E2 -13199.671} C_VEL
LIN {X 0,Y 361.947,Z 275.026,A -85,B 0,C 180,E1 -13203.474,E2 -13203.474} C_VEL
LIN {X 0,Y 361.882,Z 275.031,A -85,B 0,C 180,E1 -13207.143,E2 -13207.143} C_VEL
LIN {X 0,Y 361.912,Z 275.025,A -85,B 0,C 180,E1 -13210.723,E2 -13210.723} C_VEL
LIN {X 0,Y 361.937,Z 275.022,A -85,B 0,C 180,E1 -13214.225,E2 -13214.225} C_VEL
LIN {X 0,Y 361.99,Z 275.015,A -85,B 0,C 180,E1 -13216.527,E2 -13216.527} C_VEL
LIN {X 0,Y 362.026,Z 275.012,A -85,B 0,C 180,E1 -13219.937,E2 -13219.937} C_VEL
LIN {X 0,Y 362.14,Z 274.997,A -85,B 0,C 180,E1 -13222.192,E2 -13222.192} C_VEL
LIN {X 0,Y 362.089,Z 275.003,A -85,B 0,C 180,E1 -13224.43,E2 -13224.43} C_VEL
LIN {X 0,Y 362.052,Z 275.186,A -85,B 0,C 180,E1 -13228.887,E2 -13228.887} C_VEL
LIN {X 0,Y 361.443,Z 279.942,A -85,B 0,C 180,E1 -13234.739,E2 -13234.739} C_VEL
LIN {X 0,Y 362.462,Z 283.083,A -85,B 0,C 180,E1 -13234.935,E2 -13234.935} C_VEL
